Yaskawa INFORM job: apremTRJ0.JBI

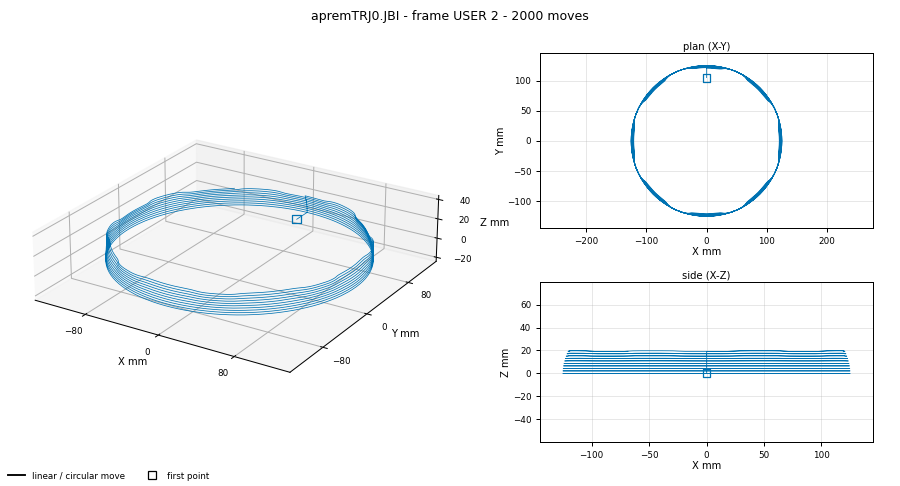
[picture p0: tool path of apremTRJ0.JBI in frame USER 2, 2000 of 2000 moves have a stored position in this frame; points joined in program order, loops and branches not executed]
/JOB
//NAME apremTRJ0
//POS
///NPOS 2000,0,0,0,0,0
///USER 2
///TOOL 1
///POSTYPE USER
///RECTAN
///RCONF 1,0,0,0,0,0,0,0,0,0,0,0,0,0,0,0,0,0,0,0,0,0,0,0
C00000=0.000,105.000,0.000,-180.0000,0.0000,0.0000
C00001=0.000,125.000,0.000,-180.0000,0.0000,0.0000
C00002=7.240,124.790,0.000,-180.0000,-0.0000,0.0000
C00003=13.736,124.243,0.000,-180.0000,-0.0000,0.0000
C00004=19.454,123.477,0.000,-180.0000,-0.0000,0.0000
C00005=23.373,122.796,0.000,-180.0000,-0.0000,0.0000
C00006=26.068,122.252,0.000,-180.0000,-0.0000,0.0000
C00007=28.242,121.768,0.000,-180.0000,-0.0000,0.0000
C00008=30.439,121.237,0.000,-180.0000,-0.0000,0.0000
C00009=33.187,120.514,0.000,-180.0000,-0.0000,0.0000
C00010=36.560,119.534,0.000,-180.0000,-0.0000,0.0000
C00011=40.117,118.388,0.000,-180.0000,-0.0000,0.0000
C00012=43.423,117.215,0.000,-180.0000,-0.0000,0.0000
C00013=46.401,116.069,0.000,-180.0000,-0.0000,0.0000
C00014=49.262,114.884,0.000,-180.0000,-0.0000,0.0000
C00015=52.179,113.589,0.000,-180.0000,-0.0000,0.0000
C00016=55.346,112.080,0.000,180.0000,0.0000,0.0000
C00017=58.672,110.375,0.000,180.0000,0.0000,0.0000
C00018=61.749,108.683,0.000,-180.0000,-0.0000,0.0000
C00019=64.204,107.252,0.000,-180.0000,-0.0000,0.0000
C00020=66.133,106.073,0.000,-180.0000,-0.0000,0.0000
C00021=68.012,104.878,0.000,-180.0000,-0.0000,0.0000
C00022=70.303,103.357,0.000,-180.0000,-0.0000,0.0000
C00023=73.555,101.068,0.000,-180.0000,-0.0000,0.0000
C00024=78.141,97.566,0.000,-180.0000,-0.0000,0.0000
C00025=83.120,93.359,0.000,-180.0000,-0.0000,0.0000
C00026=88.388,88.388,0.000,-180.0000,-0.0000,0.0000
C00027=93.359,83.120,0.000,-180.0000,-0.0000,0.0000
C00028=97.566,78.141,0.000,-180.0000,-0.0000,0.0000
C00029=101.068,73.555,0.000,180.0000,0.0000,0.0000
C00030=103.357,70.303,0.000,-180.0000,-0.0000,0.0000
C00031=104.878,68.012,0.000,-180.0000,-0.0000,0.0000
C00032=106.073,66.133,0.000,-180.0000,-0.0000,0.0000
C00033=107.252,64.204,0.000,-180.0000,-0.0000,0.0000
C00034=108.683,61.749,0.000,-180.0000,-0.0000,0.0000
C00035=110.375,58.672,0.000,-180.0000,-0.0000,0.0000
C00036=112.080,55.346,0.000,-180.0000,-0.0000,0.0000
C00037=113.589,52.179,0.000,-180.0000,-0.0000,0.0000
C00038=114.884,49.262,0.000,-180.0000,-0.0000,0.0000
C00039=116.069,46.401,0.000,-180.0000,-0.0000,0.0000
C00040=117.215,43.423,0.000,-180.0000,-0.0000,0.0000
C00041=118.388,40.117,0.000,-180.0000,-0.0000,0.0000
C00042=119.534,36.560,0.000,-180.0000,-0.0000,0.0000
C00043=120.514,33.187,0.000,-180.0000,-0.0000,0.0000
C00044=121.237,30.439,0.000,-180.0000,-0.0000,0.0000
C00045=121.768,28.242,0.000,-180.0000,-0.0000,0.0000
C00046=122.252,26.068,0.000,-180.0000,-0.0000,0.0000
C00047=122.796,23.373,0.000,-180.0000,-0.0000,0.0000
C00048=123.477,19.454,0.000,-180.0000,-0.0000,0.0000
C00049=124.243,13.736,0.000,-180.0000,-0.0000,0.0000
C00050=124.790,7.240,0.000,-180.0000,-0.0000,0.0000
C00051=125.000,0.000,0.000,-180.0000,-0.0000,0.0000
C00052=124.790,-7.240,0.000,180.0000,-0.0000,0.0000
C00053=124.243,-13.736,0.000,180.0000,-0.0000,0.0000
C00054=123.477,-19.454,0.000,180.0000,-0.0000,0.0000
C00055=122.796,-23.373,0.000,180.0000,-0.0000,0.0000
C00056=122.252,-26.068,0.000,180.0000,-0.0000,0.0000
C00057=121.768,-28.242,0.000,180.0000,-0.0000,0.0000
C00058=121.237,-30.439,0.000,180.0000,-0.0000,0.0000
C00059=120.514,-33.187,0.000,180.0000,-0.0000,0.0000
C00060=119.534,-36.560,0.000,180.0000,-0.0000,0.0000
C00061=118.388,-40.117,0.000,180.0000,-0.0000,0.0000
C00062=117.215,-43.423,0.000,180.0000,-0.0000,0.0000
C00063=116.069,-46.401,0.000,180.0000,-0.0000,0.0000
C00064=114.884,-49.262,0.000,180.0000,-0.0000,0.0000
C00065=113.589,-52.179,0.000,180.0000,-0.0000,0.0000
C00066=112.080,-55.346,0.000,180.0000,-0.0000,0.0000
C00067=110.375,-58.672,0.000,180.0000,-0.0000,0.0000
C00068=108.683,-61.749,0.000,180.0000,-0.0000,0.0000
C00069=107.252,-64.204,0.000,180.0000,-0.0000,0.0000
C00070=106.073,-66.133,0.000,180.0000,-0.0000,0.0000
C00071=104.878,-68.012,0.000,180.0000,-0.0000,0.0000
C00072=103.357,-70.303,0.000,180.0000,-0.0000,0.0000
C00073=101.068,-73.555,0.000,180.0000,-0.0000,0.0000
C00074=97.566,-78.141,0.000,180.0000,-0.0000,0.0000
C00075=93.359,-83.120,0.000,180.0000,-0.0000,0.0000
C00076=88.388,-88.388,0.000,180.0000,-0.0000,0.0000
C00077=83.120,-93.359,0.000,180.0000,-0.0000,0.0000
C00078=78.141,-97.566,0.000,180.0000,-0.0000,0.0000
C00079=73.555,-101.068,0.000,180.0000,-0.0000,0.0000
C00080=70.303,-103.357,0.000,180.0000,-0.0000,0.0000
C00081=68.012,-104.878,0.000,180.0000,-0.0000,0.0000
C00082=66.133,-106.073,0.000,180.0000,-0.0000,0.0000
C00083=64.204,-107.252,0.000,180.0000,-0.0000,0.0000
C00084=61.749,-108.683,0.000,-180.0000,0.0000,0.0000
C00085=58.672,-110.375,0.000,180.0000,-0.0000,0.0000
C00086=55.346,-112.080,0.000,180.0000,-0.0000,0.0000
C00087=52.179,-113.589,0.000,180.0000,-0.0000,0.0000
C00088=49.262,-114.884,0.000,180.0000,-0.0000,0.0000
C00089=46.401,-116.069,0.000,180.0000,-0.0000,0.0000
C00090=43.423,-117.215,0.000,180.0000,-0.0000,0.0000
C00091=40.117,-118.388,0.000,180.0000,-0.0000,0.0000
C00092=36.560,-119.534,0.000,180.0000,-0.0000,0.0000
C00093=33.187,-120.514,0.000,180.0000,-0.0000,0.0000
C00094=30.439,-121.237,0.000,180.0000,-0.0000,0.0000
C00095=28.242,-121.768,0.000,180.0000,-0.0000,0.0000
C00096=26.068,-122.252,0.000,180.0000,-0.0000,0.0000
C00097=23.373,-122.796,0.000,180.0000,-0.0000,0.0000
C00098=19.454,-123.477,0.000,180.0000,-0.0000,0.0000
C00099=13.736,-124.243,0.000,180.0000,-0.0000,0.0000
C00100=7.240,-124.790,0.000,180.0000,-0.0000,0.0000
C00101=0.000,-125.000,0.000,-180.0000,-0.0000,0.0000
C00102=0.000,-125.000,0.000,-180.0000,-0.0000,0.0000
C00103=-7.240,-124.790,0.000,-180.0000,-0.0000,0.0000
C00104=-13.736,-124.243,0.000,-180.0000,-0.0000,0.0000
C00105=-19.454,-123.477,0.000,-180.0000,-0.0000,0.0000
C00106=-23.373,-122.796,0.000,-180.0000,-0.0000,0.0000
C00107=-26.068,-122.252,0.000,-180.0000,-0.0000,0.0000
C00108=-28.242,-121.768,0.000,-180.0000,-0.0000,0.0000
C00109=-30.439,-121.237,0.000,-180.0000,-0.0000,0.0000
C00110=-33.187,-120.514,0.000,-180.0000,-0.0000,0.0000
C00111=-36.560,-119.534,0.000,-180.0000,-0.0000,0.0000
C00112=-40.117,-118.388,0.000,-180.0000,-0.0000,0.0000
C00113=-43.423,-117.215,0.000,-180.0000,-0.0000,0.0000
C00114=-46.401,-116.069,0.000,-180.0000,-0.0000,0.0000
C00115=-49.262,-114.884,0.000,-180.0000,-0.0000,0.0000
C00116=-52.179,-113.589,0.000,-180.0000,-0.0000,0.0000
C00117=-55.346,-112.080,0.000,-180.0000,-0.0000,0.0000
C00118=-58.672,-110.375,0.000,-180.0000,-0.0000,0.0000
C00119=-61.749,-108.683,0.000,-180.0000,-0.0000,0.0000
C00120=-64.204,-107.252,0.000,-180.0000,-0.0000,0.0000
C00121=-66.133,-106.073,0.000,-180.0000,-0.0000,0.0000
C00122=-68.012,-104.878,0.000,-180.0000,-0.0000,0.0000
C00123=-70.303,-103.357,0.000,-180.0000,-0.0000,0.0000
C00124=-73.555,-101.068,0.000,-180.0000,-0.0000,0.0000
C00125=-78.141,-97.566,0.000,-180.0000,-0.0000,0.0000
C00126=-83.120,-93.359,0.000,-180.0000,-0.0000,0.0000
C00127=-88.388,-88.388,0.000,-180.0000,-0.0000,0.0000
C00128=-93.359,-83.120,0.000,-180.0000,-0.0000,0.0000
C00129=-97.566,-78.141,0.000,-180.0000,-0.0000,0.0000
C00130=-101.068,-73.555,0.000,-180.0000,-0.0000,0.0000
C00131=-103.357,-70.303,0.000,-180.0000,-0.0000,0.0000
C00132=-104.878,-68.012,0.000,-180.0000,-0.0000,0.0000
C00133=-106.073,-66.133,0.000,-180.0000,-0.0000,0.0000
C00134=-107.252,-64.204,0.000,-180.0000,-0.0000,0.0000
C00135=-108.683,-61.749,0.000,-180.0000,-0.0000,0.0000
C00136=-110.375,-58.672,0.000,-180.0000,-0.0000,0.0000
C00137=-112.080,-55.346,0.000,-180.0000,-0.0000,0.0000
C00138=-113.589,-52.179,0.000,180.0000,0.0000,0.0000
C00139=-114.884,-49.262,0.000,180.0000,0.0000,0.0000
C00140=-116.069,-46.401,0.000,-180.0000,-0.0000,0.0000
C00141=-117.215,-43.423,0.000,-180.0000,-0.0000,0.0000
C00142=-118.388,-40.117,0.000,180.0000,0.0000,0.0000
C00143=-119.534,-36.560,0.000,180.0000,0.0000,0.0000
C00144=-120.514,-33.187,0.000,-180.0000,-0.0000,0.0000
C00145=-121.237,-30.439,0.000,-180.0000,-0.0000,0.0000
C00146=-121.768,-28.242,0.000,-180.0000,-0.0000,0.0000
C00147=-122.252,-26.068,0.000,-180.0000,-0.0000,0.0000
C00148=-122.796,-23.373,0.000,-180.0000,-0.0000,0.0000
C00149=-123.477,-19.454,0.000,-180.0000,-0.0000,0.0000
C00150=-124.243,-13.736,0.000,-180.0000,-0.0000,0.0000
C00151=-124.790,-7.240,0.000,-180.0000,-0.0000,0.0000
C00152=-125.000,0.000,0.000,180.0000,0.0000,0.0000
C00153=-124.790,7.240,0.000,-180.0000,0.0000,0.0000
C00154=-124.243,13.736,0.000,-180.0000,0.0000,0.0000
C00155=-123.477,19.454,0.000,-180.0000,0.0000,0.0000
C00156=-122.796,23.373,0.000,-180.0000,0.0000,0.0000
C00157=-122.252,26.068,0.000,-180.0000,0.0000,0.0000
C00158=-121.768,28.242,0.000,-180.0000,0.0000,0.0000
C00159=-121.237,30.439,0.000,-180.0000,0.0000,0.0000
C00160=-120.514,33.187,0.000,-180.0000,0.0000,0.0000
C00161=-119.534,36.560,0.000,-180.0000,0.0000,0.0000
C00162=-118.388,40.117,0.000,-180.0000,0.0000,0.0000
C00163=-117.215,43.423,0.000,-180.0000,0.0000,0.0000
C00164=-116.069,46.401,0.000,-180.0000,0.0000,0.0000
C00165=-114.884,49.262,0.000,-180.0000,0.0000,0.0000
C00166=-113.589,52.179,0.000,-180.0000,0.0000,0.0000
C00167=-112.080,55.346,0.000,-180.0000,0.0000,0.0000
C00168=-110.375,58.672,0.000,-180.0000,0.0000,0.0000
C00169=-108.683,61.749,0.000,-180.0000,0.0000,0.0000
C00170=-107.252,64.204,0.000,-180.0000,0.0000,0.0000
C00171=-106.073,66.133,0.000,-180.0000,0.0000,0.0000
C00172=-104.878,68.012,0.000,-180.0000,0.0000,0.0000
C00173=-103.357,70.303,0.000,-180.0000,0.0000,0.0000
C00174=-101.068,73.555,0.000,-180.0000,0.0000,0.0000
C00175=-97.566,78.141,0.000,-180.0000,0.0000,0.0000
C00176=-93.359,83.120,0.000,-180.0000,0.0000,0.0000
C00177=-88.388,88.388,0.000,-180.0000,0.0000,0.0000
C00178=-83.120,93.359,0.000,-180.0000,0.0000,0.0000
C00179=-78.141,97.566,0.000,-180.0000,0.0000,0.0000
C00180=-73.555,101.068,0.000,-180.0000,0.0000,0.0000
C00181=-70.303,103.357,0.000,-180.0000,0.0000,0.0000
C00182=-68.012,104.878,0.000,-180.0000,0.0000,0.0000
C00183=-66.133,106.073,0.000,-180.0000,0.0000,0.0000
C00184=-64.204,107.252,0.000,-180.0000,0.0000,0.0000
C00185=-61.749,108.683,0.000,-180.0000,0.0000,0.0000
C00186=-58.672,110.375,0.000,-180.0000,0.0000,0.0000
C00187=-55.346,112.080,0.000,-180.0000,0.0000,0.0000
C00188=-52.179,113.589,0.000,-180.0000,0.0000,0.0000
C00189=-49.262,114.884,0.000,-180.0000,0.0000,0.0000
C00190=-46.401,116.069,0.000,-180.0000,0.0000,0.0000
C00191=-43.423,117.215,0.000,-180.0000,0.0000,0.0000
C00192=-40.117,118.388,0.000,-180.0000,0.0000,0.0000
C00193=-36.560,119.534,0.000,-180.0000,0.0000,0.0000
C00194=-33.187,120.514,0.000,-180.0000,0.0000,0.0000
C00195=-30.439,121.237,0.000,-180.0000,0.0000,0.0000
C00196=-28.242,121.768,0.000,-180.0000,0.0000,0.0000
C00197=-26.068,122.252,0.000,-180.0000,0.0000,0.0000
C00198=-23.373,122.796,0.000,-180.0000,0.0000,0.0000
C00199=-19.454,123.477,0.000,-180.0000,0.0000,0.0000
C00200=-13.736,124.243,0.000,-180.0000,0.0000,0.0000
C00201=-7.240,124.790,0.000,-180.0000,0.0000,0.0000
C00202=0.000,125.000,0.000,-180.0000,0.0000,0.0000
C00203=0.000,124.937,2.199,-176.7359,0.0000,0.0000
C00204=7.234,124.727,2.199,-176.7395,-0.1900,0.0000
C00205=13.726,124.181,2.199,-176.7605,-0.3579,0.0000
C00206=19.443,123.417,2.199,-176.9022,-0.4857,0.0000
C00207=23.359,122.743,2.199,-177.2352,-0.5194,0.0000
C00208=26.053,122.209,2.200,-177.7082,-0.4785,0.0000
C00209=28.225,121.736,2.200,-178.2567,-0.3947,0.0000
C00210=30.422,121.217,2.200,-178.8064,-0.2941,0.0000
C00211=33.169,120.504,2.200,-179.2794,-0.1963,0.0000
C00212=36.543,119.532,2.200,-179.6554,-0.1047,0.0000
C00213=40.104,118.390,2.200,-179.9022,-0.0330,0.0000
C00214=43.415,117.218,2.200,-179.9844,-0.0058,0.0000
C00215=46.399,116.070,2.200,-179.9982,-0.0007,0.0000
C00216=49.265,114.882,2.200,-179.9982,-0.0008,0.0000
C00217=52.187,113.585,2.200,-179.9849,-0.0069,0.0000
C00218=55.357,112.072,2.200,-179.9075,-0.0458,0.0000
C00219=58.682,110.361,2.200,-179.6823,-0.1696,0.0000
C00220=61.755,108.663,2.200,-179.3516,-0.3707,0.0000
C00221=64.202,107.225,2.200,-178.9481,-0.6362,0.0000
C00222=66.122,106.039,2.200,-178.4882,-0.9539,0.0000
C00223=67.993,104.837,2.200,-178.0410,-1.2829,0.0000
C00224=70.275,103.309,2.199,-177.6774,-1.5889,0.0000
C00225=73.521,101.017,2.199,-177.4656,-1.8485,0.0000
C00226=78.103,97.515,2.199,-177.4554,-2.0392,0.0000
C00227=83.080,93.311,2.199,-177.5592,-2.1726,0.0000
C00228=88.344,88.344,2.199,-177.6906,-2.3094,0.0000
C00229=93.311,83.080,2.199,-177.8274,-2.4408,0.0000
C00230=97.515,78.103,2.199,-177.9608,-2.5446,0.0000
C00231=101.017,73.521,2.199,-178.1515,-2.5344,0.0000
C00232=103.309,70.275,2.199,-178.4111,-2.3226,0.0000
C00233=104.837,67.993,2.200,-178.7171,-1.9590,0.0000
C00234=106.039,66.122,2.200,-179.0461,-1.5118,0.0000
C00235=107.225,64.202,2.200,-179.3638,-1.0519,0.0000
C00236=108.663,61.755,2.200,-179.6293,-0.6484,0.0000
C00237=110.361,58.682,2.200,-179.8304,-0.3177,0.0000
C00238=112.072,55.357,2.200,-179.9542,-0.0925,0.0000
C00239=113.585,52.187,2.200,-179.9931,-0.0151,0.0000
C00240=114.882,49.265,2.200,-179.9992,-0.0018,0.0000
C00241=116.070,46.399,2.200,-179.9993,-0.0018,0.0000
C00242=117.218,43.415,2.200,-179.9942,-0.0156,0.0000
C00243=118.390,40.104,2.200,-179.9670,-0.0978,0.0000
C00244=119.532,36.543,2.200,-179.8953,-0.3446,0.0000
C00245=120.504,33.169,2.200,-179.8037,-0.7206,0.0000
C00246=121.217,30.422,2.200,-179.7059,-1.1936,0.0000
C00247=121.736,28.225,2.200,-179.6053,-1.7433,0.0000
C00248=122.209,26.053,2.200,-179.5215,-2.2918,0.0000
C00249=122.743,23.359,2.199,-179.4806,-2.7648,0.0000
C00250=123.417,19.443,2.199,-179.5143,-3.0978,0.0000
C00251=124.181,13.726,2.199,-179.6421,-3.2395,0.0000
C00252=124.727,7.234,2.199,-179.8100,-3.2605,0.0000
C00253=124.937,0.000,2.199,180.0000,-3.2641,0.0000
C00254=124.727,-7.234,2.199,179.8100,-3.2604,0.0000
C00255=124.181,-13.726,2.199,179.6421,-3.2395,0.0000
C00256=123.417,-19.443,2.199,179.5143,-3.0978,0.0000
C00257=122.743,-23.359,2.199,179.4806,-2.7648,0.0000
C00258=122.209,-26.053,2.200,179.5215,-2.2918,0.0000
C00259=121.736,-28.225,2.200,179.6053,-1.7433,0.0000
C00260=121.217,-30.422,2.200,179.7059,-1.1936,0.0000
C00261=120.504,-33.169,2.200,179.8037,-0.7206,0.0000
C00262=119.532,-36.543,2.200,179.8953,-0.3446,0.0000
C00263=118.390,-40.104,2.200,179.9670,-0.0978,0.0000
C00264=117.218,-43.415,2.200,179.9942,-0.0156,0.0000
C00265=116.070,-46.399,2.200,179.9993,-0.0018,0.0000
C00266=114.882,-49.265,2.200,179.9992,-0.0018,0.0000
C00267=113.585,-52.187,2.200,179.9931,-0.0151,0.0000
C00268=112.072,-55.357,2.200,179.9542,-0.0925,0.0000
C00269=110.361,-58.682,2.200,179.8304,-0.3177,0.0000
C00270=108.663,-61.755,2.200,179.6293,-0.6484,0.0000
C00271=107.225,-64.202,2.200,179.3638,-1.0519,0.0000
C00272=106.039,-66.122,2.200,179.0461,-1.5118,0.0000
C00273=104.837,-67.993,2.200,178.7171,-1.9590,0.0000
C00274=103.309,-70.275,2.199,178.4111,-2.3226,0.0000
C00275=101.017,-73.521,2.199,178.1515,-2.5344,0.0000
C00276=97.515,-78.103,2.199,177.9608,-2.5446,0.0000
C00277=93.311,-83.080,2.199,177.8274,-2.4408,0.0000
C00278=88.344,-88.344,2.199,177.6906,-2.3094,0.0000
C00279=83.080,-93.311,2.199,177.5592,-2.1726,0.0000
C00280=78.103,-97.515,2.199,177.4554,-2.0392,0.0000
C00281=73.521,-101.017,2.199,177.4656,-1.8485,0.0000
C00282=70.275,-103.309,2.199,177.6774,-1.5889,0.0000
C00283=67.993,-104.837,2.200,178.0410,-1.2829,0.0000
C00284=66.122,-106.039,2.200,178.4882,-0.9539,0.0000
C00285=64.202,-107.225,2.200,178.9481,-0.6362,0.0000
C00286=61.755,-108.663,2.200,179.3516,-0.3707,0.0000
C00287=58.682,-110.361,2.200,179.6823,-0.1696,0.0000
C00288=55.357,-112.072,2.200,179.9075,-0.0458,0.0000
C00289=52.187,-113.585,2.200,179.9849,-0.0069,0.0000
C00290=49.265,-114.882,2.200,179.9982,-0.0008,0.0000
C00291=46.399,-116.070,2.200,179.9982,-0.0007,0.0000
C00292=43.415,-117.218,2.200,179.9844,-0.0058,0.0000
C00293=40.104,-118.390,2.200,179.9022,-0.0330,0.0000
C00294=36.543,-119.532,2.200,179.6554,-0.1047,0.0000
C00295=33.169,-120.504,2.200,179.2794,-0.1963,0.0000
C00296=30.422,-121.217,2.200,178.8064,-0.2941,0.0000
C00297=28.225,-121.736,2.200,178.2567,-0.3947,0.0000
C00298=26.053,-122.209,2.200,177.7082,-0.4785,0.0000
C00299=23.359,-122.743,2.199,177.2352,-0.5194,0.0000
C00300=19.443,-123.417,2.199,176.9022,-0.4857,0.0000
C00301=13.726,-124.181,2.199,176.7605,-0.3579,0.0000
C00302=7.234,-124.727,2.199,176.7395,-0.1900,0.0000
C00303=0.000,-124.937,2.199,176.7359,0.0000,0.0000
C00304=0.000,-124.937,2.199,176.7359,0.0000,0.0000
C00305=-7.234,-124.727,2.199,176.7396,0.1900,0.0000
C00306=-13.726,-124.181,2.199,176.7605,0.3579,0.0000
C00307=-19.443,-123.417,2.199,176.9022,0.4857,0.0000
C00308=-23.359,-122.743,2.199,177.2352,0.5194,0.0000
C00309=-26.053,-122.209,2.200,177.7082,0.4785,0.0000
C00310=-28.225,-121.736,2.200,178.2567,0.3947,0.0000
C00311=-30.422,-121.217,2.200,178.8064,0.2941,0.0000
C00312=-33.169,-120.504,2.200,179.2794,0.1963,0.0000
C00313=-36.543,-119.532,2.200,179.6554,0.1047,0.0000
C00314=-40.104,-118.390,2.200,179.9022,0.0330,0.0000
C00315=-43.415,-117.218,2.200,179.9844,0.0058,0.0000
C00316=-46.399,-116.070,2.200,179.9982,0.0007,0.0000
C00317=-49.265,-114.882,2.200,179.9982,0.0008,0.0000
C00318=-52.187,-113.585,2.200,179.9849,0.0069,0.0000
C00319=-55.357,-112.072,2.200,179.9075,0.0458,0.0000
C00320=-58.682,-110.361,2.200,179.6823,0.1696,0.0000
C00321=-61.755,-108.663,2.200,179.3516,0.3707,0.0000
C00322=-64.202,-107.225,2.200,178.9481,0.6362,0.0000
C00323=-66.122,-106.039,2.200,178.4882,0.9539,0.0000
C00324=-67.993,-104.837,2.200,178.0410,1.2829,0.0000
C00325=-70.275,-103.309,2.199,177.6774,1.5889,0.0000
C00326=-73.521,-101.017,2.199,177.4656,1.8485,0.0000
C00327=-78.103,-97.515,2.199,177.4554,2.0392,0.0000
C00328=-83.080,-93.311,2.199,177.5592,2.1726,0.0000
C00329=-88.344,-88.344,2.199,177.6906,2.3094,0.0000
C00330=-93.311,-83.080,2.199,177.8274,2.4408,0.0000
C00331=-97.515,-78.103,2.199,177.9608,2.5446,0.0000
C00332=-101.017,-73.521,2.199,178.1515,2.5344,0.0000
C00333=-103.309,-70.275,2.199,178.4111,2.3226,0.0000
C00334=-104.837,-67.993,2.200,178.7171,1.9590,0.0000
C00335=-106.039,-66.122,2.200,179.0461,1.5118,0.0000
C00336=-107.225,-64.202,2.200,179.3638,1.0519,0.0000
C00337=-108.663,-61.755,2.200,179.6293,0.6484,0.0000
C00338=-110.361,-58.682,2.200,179.8304,0.3177,0.0000
C00339=-112.072,-55.357,2.200,179.9542,0.0925,0.0000
C00340=-113.585,-52.187,2.200,179.9931,0.0151,0.0000
C00341=-114.882,-49.265,2.200,179.9992,0.0018,0.0000
C00342=-116.070,-46.399,2.200,179.9993,0.0018,0.0000
C00343=-117.218,-43.415,2.200,179.9942,0.0156,0.0000
C00344=-118.390,-40.104,2.200,179.9670,0.0978,0.0000
C00345=-119.532,-36.543,2.200,179.8953,0.3446,0.0000
C00346=-120.504,-33.169,2.200,179.8037,0.7206,0.0000
C00347=-121.217,-30.422,2.200,179.7059,1.1936,0.0000
C00348=-121.736,-28.225,2.200,179.6053,1.7433,0.0000
C00349=-122.209,-26.053,2.200,179.5215,2.2918,0.0000
C00350=-122.743,-23.359,2.199,179.4806,2.7648,0.0000
C00351=-123.417,-19.443,2.199,179.5143,3.0978,0.0000
C00352=-124.181,-13.726,2.199,179.6421,3.2395,0.0000
C00353=-124.727,-7.234,2.199,179.8100,3.2605,0.0000
C00354=-124.937,0.000,2.199,-180.0000,3.2641,0.0000
C00355=-124.727,7.234,2.199,-179.8100,3.2604,0.0000
C00356=-124.181,13.726,2.199,-179.6421,3.2395,0.0000
C00357=-123.417,19.443,2.199,-179.5143,3.0978,0.0000
C00358=-122.743,23.359,2.199,-179.4806,2.7648,0.0000
C00359=-122.209,26.053,2.200,-179.5215,2.2918,0.0000
C00360=-121.736,28.225,2.200,-179.6053,1.7433,0.0000
C00361=-121.217,30.422,2.200,-179.7059,1.1936,0.0000
C00362=-120.504,33.169,2.200,-179.8037,0.7206,0.0000
C00363=-119.532,36.543,2.200,-179.8953,0.3446,0.0000
C00364=-118.390,40.104,2.200,-179.9670,0.0978,0.0000
C00365=-117.218,43.415,2.200,-179.9942,0.0156,0.0000
C00366=-116.070,46.399,2.200,-179.9993,0.0018,0.0000
C00367=-114.882,49.265,2.200,-179.9992,0.0018,0.0000
C00368=-113.585,52.187,2.200,-179.9931,0.0151,0.0000
C00369=-112.072,55.357,2.200,-179.9542,0.0925,0.0000
C00370=-110.361,58.682,2.200,-179.8304,0.3177,0.0000
C00371=-108.663,61.755,2.200,-179.6293,0.6484,0.0000
C00372=-107.225,64.202,2.200,-179.3638,1.0519,0.0000
C00373=-106.039,66.122,2.200,-179.0461,1.5118,0.0000
C00374=-104.837,67.993,2.200,-178.7171,1.9590,0.0000
C00375=-103.309,70.275,2.199,-178.4111,2.3226,0.0000
C00376=-101.017,73.521,2.199,-178.1515,2.5344,0.0000
C00377=-97.515,78.103,2.199,-177.9608,2.5446,0.0000
C00378=-93.311,83.080,2.199,-177.8274,2.4408,0.0000
C00379=-88.344,88.344,2.199,-177.6906,2.3094,0.0000
C00380=-83.080,93.311,2.199,-177.5592,2.1726,0.0000
C00381=-78.103,97.515,2.199,-177.4554,2.0392,0.0000
C00382=-73.521,101.017,2.199,-177.4656,1.8485,0.0000
C00383=-70.275,103.309,2.199,-177.6774,1.5889,0.0000
C00384=-67.993,104.837,2.200,-178.0410,1.2829,0.0000
C00385=-66.122,106.039,2.200,-178.4882,0.9539,0.0000
C00386=-64.202,107.225,2.200,-178.9481,0.6362,0.0000
C00387=-61.755,108.663,2.200,-179.3516,0.3707,0.0000
C00388=-58.682,110.361,2.200,-179.6823,0.1696,0.0000
C00389=-55.357,112.072,2.200,-179.9075,0.0458,0.0000
C00390=-52.187,113.585,2.200,-179.9849,0.0069,0.0000
C00391=-49.265,114.882,2.200,-179.9982,0.0008,0.0000
C00392=-46.399,116.070,2.200,-179.9982,0.0007,0.0000
C00393=-43.415,117.218,2.200,-179.9844,0.0058,0.0000
C00394=-40.104,118.390,2.200,-179.9022,0.0330,0.0000
C00395=-36.543,119.532,2.200,-179.6554,0.1047,0.0000
C00396=-33.169,120.504,2.200,-179.2794,0.1963,0.0000
C00397=-30.422,121.217,2.200,-178.8064,0.2941,0.0000
C00398=-28.225,121.736,2.200,-178.2567,0.3947,0.0000
C00399=-26.053,122.209,2.200,-177.7082,0.4785,0.0000
C00400=-23.359,122.743,2.199,-177.2352,0.5194,0.0000
C00401=-19.443,123.417,2.199,-176.9022,0.4857,0.0000
C00402=-13.726,124.181,2.199,-176.7605,0.3579,0.0000
C00403=-7.234,124.727,2.199,-176.7396,0.1900,0.0000
C00404=0.000,124.937,2.199,-176.7359,0.0000,0.0000
C00405=0.000,124.751,4.391,-173.6081,0.0000,0.0000
C00406=7.217,124.542,4.391,-173.6153,-0.3730,0.0000
C00407=13.697,123.997,4.391,-173.6559,-0.7003,0.0000
C00408=19.408,123.242,4.392,-173.9305,-0.9378,0.0000
C00409=23.317,122.588,4.393,-174.5780,-0.9792,0.0000
C00410=26.007,122.082,4.395,-175.5036,-0.8805,0.0000
C00411=28.178,121.643,4.397,-176.5830,-0.7191,0.0000
C00412=30.372,121.157,4.398,-177.6658,-0.5439,0.0000
C00413=33.115,120.475,4.399,-178.5947,-0.3708,0.0000
C00414=36.492,119.526,4.399,-179.3309,-0.1993,0.0000
C00415=40.064,118.397,4.400,-179.8118,-0.0629,0.0000
C00416=43.390,117.226,4.400,-179.9699,-0.0111,0.0000
C00417=46.390,116.073,4.400,-179.9965,-0.0014,0.0000
C00418=49.273,114.879,4.400,-179.9965,-0.0015,0.0000
C00419=52.210,113.573,4.400,-179.9709,-0.0134,0.0000
C00420=55.390,112.049,4.400,-179.8224,-0.0886,0.0000
C00421=58.714,110.321,4.399,-179.3860,-0.3322,0.0000
C00422=61.773,108.604,4.399,-178.7441,-0.7317,0.0000
C00423=64.195,107.147,4.398,-177.9648,-1.2666,0.0000
C00424=66.090,105.939,4.397,-177.0750,-1.9098,0.0000
C00425=67.935,104.715,4.395,-176.1970,-2.5616,0.0000
C00426=70.195,103.171,4.393,-175.4716,-3.1498,0.0000
C00427=73.422,100.869,4.392,-175.0413,-3.6398,0.0000
C00428=77.994,97.365,4.391,-175.0131,-4.0027,0.0000
C00429=82.961,93.168,4.391,-175.2140,-4.2618,0.0000
C00430=88.212,88.212,4.391,-175.4709,-4.5291,0.0000
C00431=93.168,82.961,4.391,-175.7382,-4.7860,0.0000
C00432=97.365,77.994,4.391,-175.9973,-4.9870,0.0000
C00433=100.869,73.422,4.392,-176.3602,-4.9586,0.0000
C00434=103.171,70.195,4.393,-176.8502,-4.5284,0.0000
C00435=104.715,67.935,4.395,-177.4384,-3.8030,0.0000
C00436=105.939,66.090,4.397,-178.0902,-2.9250,0.0000
C00437=107.147,64.195,4.398,-178.7334,-2.0352,0.0000
C00438=108.604,61.773,4.399,-179.2683,-1.2559,0.0000
C00439=110.321,58.714,4.399,-179.6678,-0.6140,0.0000
C00440=112.049,55.390,4.400,-179.9114,-0.1776,0.0000
C00441=113.573,52.210,4.400,-179.9866,-0.0291,0.0000
C00442=114.879,49.273,4.400,-179.9985,-0.0035,0.0000
C00443=116.073,46.390,4.400,-179.9986,-0.0035,0.0000
C00444=117.226,43.390,4.400,-179.9889,-0.0301,0.0000
C00445=118.397,40.064,4.400,-179.9371,-0.1882,0.0000
C00446=119.526,36.492,4.399,-179.8007,-0.6691,0.0000
C00447=120.475,33.115,4.399,-179.6292,-1.4053,0.0000
C00448=121.157,30.372,4.398,-179.4561,-2.3342,0.0000
C00449=121.643,28.178,4.397,-179.2809,-3.4170,0.0000
C00450=122.082,26.007,4.395,-179.1195,-4.4964,0.0000
C00451=122.588,23.317,4.393,-179.0208,-5.4220,0.0000
C00452=123.242,19.408,4.392,-179.0622,-6.0695,0.0000
C00453=123.997,13.697,4.391,-179.2997,-6.3441,0.0000
C00454=124.542,7.217,4.391,-179.6270,-6.3847,0.0000
C00455=124.751,0.000,4.391,180.0000,-6.3919,0.0000
C00456=124.542,-7.217,4.391,179.6271,-6.3846,0.0000
C00457=123.997,-13.697,4.391,179.2997,-6.3441,0.0000
C00458=123.242,-19.408,4.392,179.0622,-6.0694,0.0000
C00459=122.588,-23.317,4.393,179.0208,-5.4220,0.0000
C00460=122.082,-26.007,4.395,179.1195,-4.4964,0.0000
C00461=121.643,-28.178,4.397,179.2809,-3.4170,0.0000
C00462=121.157,-30.372,4.398,179.4561,-2.3342,0.0000
C00463=120.475,-33.115,4.399,179.6292,-1.4053,0.0000
C00464=119.526,-36.492,4.399,179.8007,-0.6691,0.0000
C00465=118.397,-40.064,4.400,179.9371,-0.1882,0.0000
C00466=117.226,-43.390,4.400,179.9889,-0.0301,0.0000
C00467=116.073,-46.390,4.400,179.9986,-0.0035,0.0000
C00468=114.879,-49.273,4.400,179.9985,-0.0035,0.0000
C00469=113.573,-52.210,4.400,179.9866,-0.0291,0.0000
C00470=112.049,-55.390,4.400,179.9114,-0.1776,0.0000
C00471=110.321,-58.714,4.399,179.6678,-0.6140,0.0000
C00472=108.604,-61.773,4.399,179.2683,-1.2559,0.0000
C00473=107.147,-64.195,4.398,178.7334,-2.0352,0.0000
C00474=105.939,-66.090,4.397,178.0902,-2.9250,0.0000
C00475=104.715,-67.935,4.395,177.4384,-3.8030,0.0000
C00476=103.171,-70.195,4.393,176.8502,-4.5284,0.0000
C00477=100.869,-73.422,4.392,176.3602,-4.9587,0.0000
C00478=97.365,-77.994,4.391,175.9973,-4.9869,0.0000
C00479=93.168,-82.961,4.391,175.7382,-4.7860,0.0000
C00480=88.212,-88.212,4.391,175.4709,-4.5291,0.0000
C00481=82.961,-93.168,4.391,175.2140,-4.2618,0.0000
C00482=77.994,-97.365,4.391,175.0130,-4.0027,0.0000
C00483=73.422,-100.869,4.392,175.0414,-3.6398,0.0000
C00484=70.195,-103.171,4.393,175.4716,-3.1498,0.0000
C00485=67.935,-104.715,4.395,176.1970,-2.5616,0.0000
C00486=66.090,-105.939,4.397,177.0750,-1.9098,0.0000
C00487=64.195,-107.147,4.398,177.9648,-1.2666,0.0000
C00488=61.773,-108.604,4.399,178.7441,-0.7317,0.0000
C00489=58.714,-110.321,4.399,179.3860,-0.3322,0.0000
C00490=55.390,-112.049,4.400,179.8224,-0.0886,0.0000
C00491=52.210,-113.573,4.400,179.9709,-0.0134,0.0000
C00492=49.273,-114.879,4.400,179.9965,-0.0015,0.0000
C00493=46.390,-116.073,4.400,179.9965,-0.0014,0.0000
C00494=43.390,-117.226,4.400,179.9699,-0.0111,0.0000
C00495=40.064,-118.397,4.400,179.8118,-0.0629,0.0000
C00496=36.492,-119.526,4.399,179.3309,-0.1993,0.0000
C00497=33.115,-120.475,4.399,178.5947,-0.3708,0.0000
C00498=30.372,-121.157,4.398,177.6658,-0.5439,0.0000
C00499=28.178,-121.643,4.397,176.5830,-0.7191,0.0000
C00500=26.007,-122.082,4.395,175.5036,-0.8805,0.0000
C00501=23.317,-122.588,4.393,174.5780,-0.9792,0.0000
C00502=19.408,-123.242,4.392,173.9305,-0.9378,0.0000
C00503=13.697,-123.997,4.391,173.6559,-0.7003,0.0000
C00504=7.217,-124.542,4.391,173.6153,-0.3730,0.0000
C00505=0.000,-124.751,4.391,173.6081,0.0000,0.0000
C00506=0.000,-124.751,4.391,173.6081,0.0000,0.0000
C00507=-7.217,-124.542,4.391,173.6154,0.3729,0.0000
C00508=-13.697,-123.997,4.391,173.6559,0.7003,0.0000
C00509=-19.408,-123.242,4.392,173.9306,0.9378,0.0000
C00510=-23.317,-122.588,4.393,174.5780,0.9792,0.0000
C00511=-26.007,-122.082,4.395,175.5036,0.8805,0.0000
C00512=-28.178,-121.643,4.397,176.5830,0.7191,0.0000
C00513=-30.372,-121.157,4.398,177.6658,0.5439,0.0000
C00514=-33.115,-120.475,4.399,178.5947,0.3708,0.0000
C00515=-36.492,-119.526,4.399,179.3309,0.1993,0.0000
C00516=-40.064,-118.397,4.400,179.8118,0.0629,0.0000
C00517=-43.390,-117.226,4.400,179.9699,0.0111,0.0000
C00518=-46.390,-116.073,4.400,179.9965,0.0014,0.0000
C00519=-49.273,-114.879,4.400,179.9965,0.0015,0.0000
C00520=-52.210,-113.573,4.400,179.9709,0.0134,0.0000
C00521=-55.390,-112.049,4.400,179.8224,0.0886,0.0000
C00522=-58.714,-110.321,4.399,179.3860,0.3322,0.0000
C00523=-61.773,-108.604,4.399,178.7441,0.7317,0.0000
C00524=-64.195,-107.147,4.398,177.9648,1.2666,0.0000
C00525=-66.090,-105.939,4.397,177.0750,1.9098,0.0000
C00526=-67.935,-104.715,4.395,176.1970,2.5616,0.0000
C00527=-70.195,-103.171,4.393,175.4716,3.1498,0.0000
C00528=-73.422,-100.869,4.392,175.0413,3.6398,0.0000
C00529=-77.994,-97.365,4.391,175.0131,4.0027,0.0000
C00530=-82.961,-93.168,4.391,175.2140,4.2618,0.0000
C00531=-88.212,-88.212,4.391,175.4709,4.5291,0.0000
C00532=-93.168,-82.961,4.391,175.7382,4.7860,0.0000
C00533=-97.365,-77.994,4.391,175.9973,4.9870,0.0000
C00534=-100.869,-73.422,4.392,176.3602,4.9586,0.0000
C00535=-103.171,-70.195,4.393,176.8502,4.5284,0.0000
C00536=-104.715,-67.935,4.395,177.4384,3.8030,0.0000
C00537=-105.939,-66.090,4.397,178.0902,2.9250,0.0000
C00538=-107.147,-64.195,4.398,178.7334,2.0352,0.0000
C00539=-108.604,-61.773,4.399,179.2683,1.2559,0.0000
C00540=-110.321,-58.714,4.399,179.6678,0.6140,0.0000
C00541=-112.049,-55.390,4.400,179.9114,0.1776,0.0000
C00542=-113.573,-52.210,4.400,179.9866,0.0291,0.0000
C00543=-114.879,-49.273,4.400,179.9985,0.0035,0.0000
C00544=-116.073,-46.390,4.400,179.9986,0.0035,0.0000
C00545=-117.226,-43.390,4.400,179.9889,0.0301,0.0000
C00546=-118.397,-40.064,4.400,179.9371,0.1882,0.0000
C00547=-119.526,-36.492,4.399,179.8007,0.6691,0.0000
C00548=-120.475,-33.115,4.399,179.6292,1.4053,0.0000
C00549=-121.157,-30.372,4.398,179.4561,2.3342,0.0000
C00550=-121.643,-28.178,4.397,179.2809,3.4170,0.0000
C00551=-122.082,-26.007,4.395,179.1195,4.4964,0.0000
C00552=-122.588,-23.317,4.393,179.0208,5.4220,0.0000
C00553=-123.242,-19.408,4.392,179.0622,6.0695,0.0000
C00554=-123.997,-13.697,4.391,179.2997,6.3441,0.0000
C00555=-124.542,-7.217,4.391,179.6270,6.3847,0.0000
C00556=-124.751,0.000,4.391,-180.0000,6.3919,0.0000
C00557=-124.542,7.217,4.391,-179.6271,6.3846,0.0000
C00558=-123.997,13.697,4.391,-179.2997,6.3441,0.0000
C00559=-123.242,19.408,4.392,-179.0622,6.0694,0.0000
C00560=-122.588,23.317,4.393,-179.0208,5.4220,0.0000
C00561=-122.082,26.007,4.395,-179.1195,4.4964,0.0000
C00562=-121.643,28.178,4.397,-179.2809,3.4170,0.0000
C00563=-121.157,30.372,4.398,-179.4561,2.3342,0.0000
C00564=-120.475,33.115,4.399,-179.6292,1.4053,0.0000
C00565=-119.526,36.492,4.399,-179.8007,0.6691,0.0000
C00566=-118.397,40.064,4.400,-179.9371,0.1882,0.0000
C00567=-117.226,43.390,4.400,-179.9889,0.0301,0.0000
C00568=-116.073,46.390,4.400,-179.9986,0.0035,0.0000
C00569=-114.879,49.273,4.400,-179.9985,0.0035,0.0000
C00570=-113.573,52.210,4.400,-179.9866,0.0291,0.0000
C00571=-112.049,55.390,4.400,-179.9114,0.1776,0.0000
C00572=-110.321,58.714,4.399,-179.6678,0.6140,0.0000
C00573=-108.604,61.773,4.399,-179.2683,1.2559,0.0000
C00574=-107.147,64.195,4.398,-178.7334,2.0352,0.0000
C00575=-105.939,66.090,4.397,-178.0902,2.9250,0.0000
C00576=-104.715,67.935,4.395,-177.4384,3.8030,0.0000
C00577=-103.171,70.195,4.393,-176.8502,4.5284,0.0000
C00578=-100.869,73.422,4.392,-176.3602,4.9587,0.0000
C00579=-97.365,77.994,4.391,-175.9973,4.9869,0.0000
C00580=-93.168,82.961,4.391,-175.7382,4.7860,0.0000
C00581=-88.212,88.212,4.391,-175.4709,4.5291,0.0000
C00582=-82.961,93.168,4.391,-175.2140,4.2618,0.0000
C00583=-77.994,97.365,4.391,-175.0130,4.0027,0.0000
C00584=-73.422,100.869,4.392,-175.0414,3.6398,0.0000
C00585=-70.195,103.171,4.393,-175.4716,3.1498,0.0000
C00586=-67.935,104.715,4.395,-176.1970,2.5616,0.0000
C00587=-66.090,105.939,4.397,-177.0750,1.9098,0.0000
C00588=-64.195,107.147,4.398,-177.9648,1.2666,0.0000
C00589=-61.773,108.604,4.399,-178.7441,0.7317,0.0000
C00590=-58.714,110.321,4.399,-179.3860,0.3322,0.0000
C00591=-55.390,112.049,4.400,-179.8224,0.0886,0.0000
C00592=-52.210,113.573,4.400,-179.9709,0.0134,0.0000
C00593=-49.273,114.879,4.400,-179.9965,0.0015,0.0000
C00594=-46.390,116.073,4.400,-179.9965,0.0014,0.0000
C00595=-43.390,117.226,4.400,-179.9699,0.0111,0.0000
C00596=-40.064,118.397,4.400,-179.8118,0.0629,0.0000
C00597=-36.492,119.526,4.399,-179.3309,0.1993,0.0000
C00598=-33.115,120.475,4.399,-178.5947,0.3708,0.0000
C00599=-30.372,121.157,4.398,-177.6658,0.5439,0.0000
C00600=-28.178,121.643,4.397,-176.5830,0.7191,0.0000
C00601=-26.007,122.082,4.395,-175.5036,0.8805,0.0000
C00602=-23.317,122.588,4.393,-174.5780,0.9792,0.0000
C00603=-19.408,123.242,4.392,-173.9306,0.9378,0.0000
C00604=-13.697,123.997,4.391,-173.6559,0.7003,0.0000
C00605=-7.217,124.542,4.391,-173.6154,0.3729,0.0000
C00606=0.000,124.751,4.391,-173.6081,0.0000,0.0000
C00607=0.000,124.449,6.570,-170.6405,0.0000,0.0000
C00608=7.190,124.241,6.570,-170.6509,-0.5483,0.0000
C00609=13.651,123.699,6.570,-170.7093,-1.0235,0.0000
C00610=19.352,122.957,6.573,-171.1043,-1.3408,0.0000
C00611=23.250,122.335,6.578,-172.0415,-1.3416,0.0000
C00612=25.933,121.876,6.584,-173.3969,-1.1521,0.0000
C00613=28.099,121.490,6.590,-174.9904,-0.9229,0.0000
C00614=30.290,121.060,6.595,-176.5889,-0.7201,0.0000
C00615=33.027,120.427,6.597,-177.9550,-0.5107,0.0000
C00616=36.409,119.516,6.598,-179.0332,-0.2787,0.0000
C00617=39.998,118.409,6.599,-179.7323,-0.0880,0.0000
C00618=43.349,117.240,6.599,-179.9569,-0.0159,0.0000
C00619=46.376,116.078,6.600,-179.9949,-0.0020,0.0000
C00620=49.287,114.873,6.600,-179.9950,-0.0021,0.0000
C00621=52.249,113.553,6.599,-179.9583,-0.0192,0.0000
C00622=55.445,112.011,6.599,-179.7485,-0.1271,0.0000
C00623=58.765,110.256,6.598,-179.1193,-0.4866,0.0000
C00624=61.801,108.508,6.597,-178.1928,-1.0854,0.0000
C00625=64.184,107.020,6.595,-177.0785,-1.9049,0.0000
C00626=66.037,105.776,6.590,-175.8035,-2.8963,0.0000
C00627=67.842,104.516,6.584,-174.5122,-3.8692,0.0000
C00628=70.064,102.945,6.578,-173.4163,-4.7046,0.0000
C00629=73.260,100.628,6.573,-172.7494,-5.3772,0.0000
C00630=77.816,97.121,6.570,-172.6884,-5.8831,0.0000
C00631=82.768,92.936,6.570,-172.9775,-6.2574,0.0000
C00632=87.999,87.999,6.570,-173.3523,-6.6477,0.0000
C00633=92.936,82.768,6.570,-173.7426,-7.0224,0.0000
C00634=97.121,77.816,6.570,-174.1168,-7.3116,0.0000
C00635=100.628,73.260,6.573,-174.6229,-7.2506,0.0000
C00636=102.945,70.064,6.578,-175.2954,-6.5837,0.0000
C00637=104.516,67.842,6.584,-176.1308,-5.4878,0.0000
C00638=105.776,66.037,6.590,-177.1037,-4.1965,0.0000
C00639=107.020,64.184,6.595,-178.0951,-2.9215,0.0000
C00640=108.508,61.801,6.597,-178.9146,-1.8072,0.0000
C00641=110.256,58.765,6.598,-179.5134,-0.8807,0.0000
C00642=112.011,55.445,6.599,-179.8729,-0.2515,0.0000
C00643=113.553,52.249,6.599,-179.9808,-0.0417,0.0000
C00644=114.873,49.287,6.600,-179.9979,-0.0050,0.0000
C00645=116.078,46.376,6.600,-179.9980,-0.0051,0.0000
C00646=117.240,43.349,6.599,-179.9841,-0.0431,0.0000
C00647=118.409,39.998,6.599,-179.9120,-0.2677,0.0000
C00648=119.516,36.409,6.598,-179.7213,-0.9668,0.0000
C00649=120.427,33.027,6.597,-179.4893,-2.0450,0.0000
C00650=121.060,30.290,6.595,-179.2799,-3.4111,0.0000
C00651=121.490,28.099,6.590,-179.0771,-5.0096,0.0000
C00652=121.876,25.933,6.584,-178.8479,-6.6031,0.0000
C00653=122.335,23.250,6.578,-178.6584,-7.9585,0.0000
C00654=122.957,19.352,6.573,-178.6592,-8.8957,0.0000
C00655=123.699,13.651,6.570,-178.9765,-9.2907,0.0000
C00656=124.241,7.190,6.570,-179.4517,-9.3491,0.0000
C00657=124.449,0.000,6.570,180.0000,-9.3595,0.0000
C00658=124.241,-7.190,6.570,179.4517,-9.3491,0.0000
C00659=123.699,-13.651,6.570,178.9765,-9.2907,0.0000
C00660=122.957,-19.352,6.573,178.6592,-8.8957,0.0000
C00661=122.335,-23.250,6.578,178.6584,-7.9585,0.0000
C00662=121.876,-25.933,6.584,178.8479,-6.6031,0.0000
C00663=121.490,-28.099,6.590,179.0771,-5.0096,0.0000
C00664=121.060,-30.290,6.595,179.2799,-3.4111,0.0000
C00665=120.427,-33.027,6.597,179.4893,-2.0450,0.0000
C00666=119.516,-36.409,6.598,179.7213,-0.9668,0.0000
C00667=118.409,-39.998,6.599,179.9120,-0.2677,0.0000
C00668=117.240,-43.349,6.599,179.9841,-0.0431,0.0000
C00669=116.078,-46.376,6.600,179.9980,-0.0051,0.0000
C00670=114.873,-49.287,6.600,179.9979,-0.0050,0.0000
C00671=113.553,-52.249,6.599,179.9808,-0.0417,0.0000
C00672=112.011,-55.445,6.599,179.8729,-0.2515,0.0000
C00673=110.256,-58.765,6.598,179.5134,-0.8807,0.0000
C00674=108.508,-61.801,6.597,178.9146,-1.8072,0.0000
C00675=107.020,-64.184,6.595,178.0951,-2.9215,0.0000
C00676=105.776,-66.037,6.590,177.1037,-4.1965,0.0000
C00677=104.516,-67.842,6.584,176.1308,-5.4878,0.0000
C00678=102.945,-70.064,6.578,175.2954,-6.5837,0.0000
C00679=100.628,-73.260,6.573,174.6228,-7.2506,0.0000
C00680=97.121,-77.816,6.570,174.1169,-7.3116,0.0000
C00681=92.936,-82.768,6.570,173.7426,-7.0225,0.0000
C00682=87.999,-87.999,6.570,173.3523,-6.6477,0.0000
C00683=82.768,-92.936,6.570,172.9776,-6.2574,0.0000
C00684=77.816,-97.121,6.570,172.6884,-5.8832,0.0000
C00685=73.260,-100.628,6.573,172.7494,-5.3771,0.0000
C00686=70.064,-102.945,6.578,173.4163,-4.7046,0.0000
C00687=67.842,-104.516,6.584,174.5122,-3.8692,0.0000
C00688=66.037,-105.776,6.590,175.8035,-2.8963,0.0000
C00689=64.184,-107.020,6.595,177.0785,-1.9049,0.0000
C00690=61.801,-108.508,6.597,178.1928,-1.0854,0.0000
C00691=58.765,-110.256,6.598,179.1193,-0.4866,0.0000
C00692=55.445,-112.011,6.599,179.7485,-0.1271,0.0000
C00693=52.249,-113.553,6.599,179.9583,-0.0192,0.0000
C00694=49.287,-114.873,6.600,179.9950,-0.0021,0.0000
C00695=46.376,-116.078,6.600,179.9949,-0.0020,0.0000
C00696=43.349,-117.240,6.599,179.9569,-0.0159,0.0000
C00697=39.998,-118.409,6.599,179.7323,-0.0880,0.0000
C00698=36.409,-119.516,6.598,179.0332,-0.2787,0.0000
C00699=33.027,-120.427,6.597,177.9550,-0.5107,0.0000
C00700=30.290,-121.060,6.595,176.5889,-0.7201,0.0000
C00701=28.099,-121.490,6.590,174.9904,-0.9229,0.0000
C00702=25.933,-121.876,6.584,173.3969,-1.1521,0.0000
C00703=23.250,-122.335,6.578,172.0415,-1.3416,0.0000
C00704=19.352,-122.957,6.573,171.1043,-1.3408,0.0000
C00705=13.651,-123.699,6.570,170.7093,-1.0235,0.0000
C00706=7.190,-124.241,6.570,170.6509,-0.5483,0.0000
C00707=0.000,-124.449,6.570,170.6405,0.0000,0.0000
C00708=0.000,-124.449,6.570,170.6405,0.0000,0.0000
C00709=-7.190,-124.241,6.570,170.6509,0.5483,0.0000
C00710=-13.651,-123.699,6.570,170.7093,1.0235,0.0000
C00711=-19.352,-122.957,6.573,171.1043,1.3408,0.0000
C00712=-23.250,-122.335,6.578,172.0415,1.3416,0.0000
C00713=-25.933,-121.876,6.584,173.3969,1.1521,0.0000
C00714=-28.099,-121.490,6.590,174.9904,0.9229,0.0000
C00715=-30.290,-121.060,6.595,176.5889,0.7201,0.0000
C00716=-33.027,-120.427,6.597,177.9550,0.5107,0.0000
C00717=-36.409,-119.516,6.598,179.0332,0.2787,0.0000
C00718=-39.998,-118.409,6.599,179.7323,0.0880,0.0000
C00719=-43.349,-117.240,6.599,179.9569,0.0159,0.0000
C00720=-46.376,-116.078,6.600,179.9949,0.0020,0.0000
C00721=-49.287,-114.873,6.600,179.9950,0.0021,0.0000
C00722=-52.249,-113.553,6.599,179.9583,0.0192,0.0000
C00723=-55.445,-112.011,6.599,179.7485,0.1271,0.0000
C00724=-58.765,-110.256,6.598,179.1193,0.4866,0.0000
C00725=-61.801,-108.508,6.597,178.1928,1.0854,0.0000
C00726=-64.184,-107.020,6.595,177.0785,1.9049,0.0000
C00727=-66.037,-105.776,6.590,175.8035,2.8963,0.0000
C00728=-67.842,-104.516,6.584,174.5122,3.8692,0.0000
C00729=-70.064,-102.945,6.578,173.4163,4.7046,0.0000
C00730=-73.260,-100.628,6.573,172.7494,5.3772,0.0000
C00731=-77.816,-97.121,6.570,172.6884,5.8831,0.0000
C00732=-82.768,-92.936,6.570,172.9775,6.2574,0.0000
C00733=-87.999,-87.999,6.570,173.3523,6.6477,0.0000
C00734=-92.936,-82.768,6.570,173.7426,7.0224,0.0000
C00735=-97.121,-77.816,6.570,174.1168,7.3116,0.0000
C00736=-100.628,-73.260,6.573,174.6229,7.2506,0.0000
C00737=-102.945,-70.064,6.578,175.2954,6.5837,0.0000
C00738=-104.516,-67.842,6.584,176.1308,5.4878,0.0000
C00739=-105.776,-66.037,6.590,177.1037,4.1965,0.0000
C00740=-107.020,-64.184,6.595,178.0951,2.9215,0.0000
C00741=-108.508,-61.801,6.597,178.9146,1.8072,0.0000
C00742=-110.256,-58.765,6.598,179.5134,0.8807,0.0000
C00743=-112.011,-55.445,6.599,179.8729,0.2515,0.0000
C00744=-113.553,-52.249,6.599,179.9808,0.0417,0.0000
C00745=-114.873,-49.287,6.600,179.9979,0.0050,0.0000
C00746=-116.078,-46.376,6.600,179.9980,0.0051,0.0000
C00747=-117.240,-43.349,6.599,179.9841,0.0431,0.0000
C00748=-118.409,-39.998,6.599,179.9120,0.2677,0.0000
C00749=-119.516,-36.409,6.598,179.7213,0.9668,0.0000
C00750=-120.427,-33.027,6.597,179.4893,2.0450,0.0000
C00751=-121.060,-30.290,6.595,179.2799,3.4111,0.0000
C00752=-121.490,-28.099,6.590,179.0771,5.0096,0.0000
C00753=-121.876,-25.933,6.584,178.8479,6.6031,0.0000
C00754=-122.335,-23.250,6.578,178.6584,7.9585,0.0000
C00755=-122.957,-19.352,6.573,178.6592,8.8957,0.0000
C00756=-123.699,-13.651,6.570,178.9765,9.2907,0.0000
C00757=-124.241,-7.190,6.570,179.4517,9.3491,0.0000
C00758=-124.449,0.000,6.570,-180.0000,9.3595,0.0000
C00759=-124.241,7.190,6.570,-179.4517,9.3491,0.0000
C00760=-123.699,13.651,6.570,-178.9765,9.2907,0.0000
C00761=-122.957,19.352,6.573,-178.6592,8.8957,0.0000
C00762=-122.335,23.250,6.578,-178.6584,7.9585,0.0000
C00763=-121.876,25.933,6.584,-178.8479,6.6031,0.0000
C00764=-121.490,28.099,6.590,-179.0771,5.0096,0.0000
C00765=-121.060,30.290,6.595,-179.2799,3.4111,0.0000
C00766=-120.427,33.027,6.597,-179.4893,2.0450,0.0000
C00767=-119.516,36.409,6.598,-179.7213,0.9668,0.0000
C00768=-118.409,39.998,6.599,-179.9120,0.2677,0.0000
C00769=-117.240,43.349,6.599,-179.9841,0.0431,0.0000
C00770=-116.078,46.376,6.600,-179.9980,0.0051,0.0000
C00771=-114.873,49.287,6.600,-179.9979,0.0050,0.0000
C00772=-113.553,52.249,6.599,-179.9808,0.0417,0.0000
C00773=-112.011,55.445,6.599,-179.8729,0.2515,0.0000
C00774=-110.256,58.765,6.598,-179.5134,0.8807,0.0000
C00775=-108.508,61.801,6.597,-178.9146,1.8072,0.0000
C00776=-107.020,64.184,6.595,-178.0951,2.9215,0.0000
C00777=-105.776,66.037,6.590,-177.1037,4.1965,0.0000
C00778=-104.516,67.842,6.584,-176.1308,5.4878,0.0000
C00779=-102.945,70.064,6.578,-175.2954,6.5837,0.0000
C00780=-100.628,73.260,6.573,-174.6228,7.2506,0.0000
C00781=-97.121,77.816,6.570,-174.1169,7.3116,0.0000
C00782=-92.936,82.768,6.570,-173.7426,7.0225,0.0000
C00783=-87.999,87.999,6.570,-173.3523,6.6477,0.0000
C00784=-82.768,92.936,6.570,-172.9776,6.2574,0.0000
C00785=-77.816,97.121,6.570,-172.6884,5.8832,0.0000
C00786=-73.260,100.628,6.573,-172.7494,5.3771,0.0000
C00787=-70.064,102.945,6.578,-173.4163,4.7046,0.0000
C00788=-67.842,104.516,6.584,-174.5122,3.8692,0.0000
C00789=-66.037,105.776,6.590,-175.8035,2.8963,0.0000
C00790=-64.184,107.020,6.595,-177.0785,1.9049,0.0000
C00791=-61.801,108.508,6.597,-178.1928,1.0854,0.0000
C00792=-58.765,110.256,6.598,-179.1193,0.4866,0.0000
C00793=-55.445,112.011,6.599,-179.7485,0.1271,0.0000
C00794=-52.249,113.553,6.599,-179.9583,0.0192,0.0000
C00795=-49.287,114.873,6.600,-179.9950,0.0021,0.0000
C00796=-46.376,116.078,6.600,-179.9949,0.0020,0.0000
C00797=-43.349,117.240,6.599,-179.9569,0.0159,0.0000
C00798=-39.998,118.409,6.599,-179.7323,0.0880,0.0000
C00799=-36.409,119.516,6.598,-179.0332,0.2787,0.0000
C00800=-33.027,120.427,6.597,-177.9550,0.5107,0.0000
C00801=-30.290,121.060,6.595,-176.5889,0.7201,0.0000
C00802=-28.099,121.490,6.590,-174.9904,0.9229,0.0000
C00803=-25.933,121.876,6.584,-173.3969,1.1521,0.0000
C00804=-23.250,122.335,6.578,-172.0415,1.3416,0.0000
C00805=-19.352,122.957,6.573,-171.1043,1.3408,0.0000
C00806=-13.651,123.699,6.570,-170.7093,1.0235,0.0000
C00807=-7.190,124.241,6.570,-170.6509,0.5483,0.0000
C00808=0.000,124.449,6.570,-170.6405,0.0000,0.0000
C00809=0.000,124.038,8.732,-167.8485,0.0000,0.0000
C00810=7.152,123.831,8.732,-167.8618,-0.7157,0.0000
C00811=13.588,123.293,8.732,-167.9360,-1.3249,0.0000
C00812=19.275,122.569,8.737,-168.4366,-1.6816,0.0000
C00813=23.159,121.990,8.749,-169.6379,-1.5733,0.0000
C00814=25.831,121.593,8.764,-171.4049,-1.2455,0.0000
C00815=27.992,121.281,8.778,-173.4987,-0.9622,0.0000
C00816=30.178,120.926,8.788,-175.5907,-0.7974,0.0000
C00817=32.905,120.361,8.792,-177.3695,-0.6059,0.0000
C00818=36.296,119.502,8.795,-178.7682,-0.3390,0.0000
C00819=39.909,118.425,8.797,-179.6664,-0.1072,0.0000
C00820=43.292,117.258,8.799,-179.9456,-0.0200,0.0000
C00821=46.357,116.086,8.800,-179.9937,-0.0025,0.0000
C00822=49.306,114.864,8.800,-179.9937,-0.0027,0.0000
C00823=52.302,113.527,8.799,-179.9474,-0.0243,0.0000
C00824=55.520,111.959,8.797,-179.6883,-0.1601,0.0000
C00825=58.836,110.166,8.795,-178.8893,-0.6314,0.0000
C00826=61.840,108.375,8.792,-177.7114,-1.4326,0.0000
C00827=64.169,106.846,8.788,-176.3172,-2.5584,0.0000
C00828=65.965,105.552,8.778,-174.7177,-3.9303,0.0000
C00829=67.714,104.245,8.764,-173.0301,-5.2283,0.0000
C00830=69.884,102.636,8.749,-171.5412,-6.2701,0.0000
C00831=73.040,100.299,8.737,-170.6062,-7.0640,0.0000
C00832=77.573,96.789,8.732,-170.4923,-7.6756,0.0000
C00833=82.504,92.619,8.732,-170.8586,-8.1522,0.0000
C00834=87.708,87.708,8.732,-171.3429,-8.6571,0.0000
C00835=92.619,82.504,8.732,-171.8478,-9.1414,0.0000
C00836=96.789,77.573,8.732,-172.3244,-9.5077,0.0000
C00837=100.299,73.040,8.737,-172.9360,-9.3937,0.0000
C00838=102.636,69.884,8.749,-173.7299,-8.4588,0.0000
C00839=104.245,67.714,8.764,-174.7717,-6.9699,0.0000
C00840=105.552,65.965,8.778,-176.0697,-5.2823,0.0000
C00841=106.846,64.169,8.788,-177.4416,-3.6828,0.0000
C00842=108.375,61.840,8.792,-178.5674,-2.2886,0.0000
C00843=110.166,58.836,8.795,-179.3686,-1.1107,0.0000
C00844=111.959,55.520,8.797,-179.8399,-0.3117,0.0000
C00845=113.527,52.302,8.799,-179.9757,-0.0526,0.0000
C00846=114.864,49.306,8.800,-179.9973,-0.0063,0.0000
C00847=116.086,46.357,8.800,-179.9975,-0.0063,0.0000
C00848=117.258,43.292,8.799,-179.9800,-0.0544,0.0000
C00849=118.425,39.909,8.797,-179.8928,-0.3336,0.0000
C00850=119.502,36.296,8.795,-179.6610,-1.2318,0.0000
C00851=120.361,32.905,8.792,-179.3941,-2.6305,0.0000
C00852=120.926,30.178,8.788,-179.2026,-4.4093,0.0000
C00853=121.281,27.992,8.778,-179.0378,-6.5013,0.0000
C00854=121.593,25.831,8.764,-178.7545,-8.5951,0.0000
C00855=121.990,23.159,8.749,-178.4267,-10.3621,0.0000
C00856=122.569,19.275,8.737,-178.3184,-11.5634,0.0000
C00857=123.293,13.588,8.732,-178.6751,-12.0640,0.0000
C00858=123.831,7.152,8.732,-179.2843,-12.1382,0.0000
C00859=124.038,0.000,8.732,180.0000,-12.1515,0.0000
C00860=123.831,-7.152,8.732,179.2844,-12.1381,0.0000
C00861=123.293,-13.588,8.732,178.6751,-12.0640,0.0000
C00862=122.569,-19.275,8.737,178.3184,-11.5634,0.0000
C00863=121.990,-23.159,8.749,178.4267,-10.3621,0.0000
C00864=121.593,-25.831,8.764,178.7545,-8.5951,0.0000
C00865=121.281,-27.992,8.778,179.0378,-6.5013,0.0000
C00866=120.926,-30.178,8.788,179.2026,-4.4093,0.0000
C00867=120.361,-32.905,8.792,179.3941,-2.6305,0.0000
C00868=119.502,-36.296,8.795,179.6610,-1.2318,0.0000
C00869=118.425,-39.909,8.797,179.8928,-0.3336,0.0000
C00870=117.258,-43.292,8.799,179.9800,-0.0544,0.0000
C00871=116.086,-46.357,8.800,179.9975,-0.0063,0.0000
C00872=114.864,-49.306,8.800,179.9973,-0.0063,0.0000
C00873=113.527,-52.302,8.799,179.9757,-0.0526,0.0000
C00874=111.959,-55.520,8.797,179.8399,-0.3117,0.0000
C00875=110.166,-58.836,8.795,179.3686,-1.1107,0.0000
C00876=108.375,-61.840,8.792,178.5674,-2.2886,0.0000
C00877=106.846,-64.169,8.788,177.4416,-3.6828,0.0000
C00878=105.552,-65.965,8.778,176.0697,-5.2823,0.0000
C00879=104.245,-67.714,8.764,174.7717,-6.9699,0.0000
C00880=102.636,-69.884,8.749,173.7299,-8.4588,0.0000
C00881=100.299,-73.040,8.737,172.9360,-9.3938,0.0000
C00882=96.789,-77.573,8.732,172.3244,-9.5077,0.0000
C00883=92.619,-82.504,8.732,171.8478,-9.1414,0.0000
C00884=87.708,-87.708,8.732,171.3429,-8.6571,0.0000
C00885=82.504,-92.619,8.732,170.8586,-8.1522,0.0000
C00886=77.573,-96.789,8.732,170.4923,-7.6756,0.0000
C00887=73.040,-100.299,8.737,170.6063,-7.0640,0.0000
C00888=69.884,-102.636,8.749,171.5412,-6.2701,0.0000
C00889=67.714,-104.245,8.764,173.0301,-5.2283,0.0000
C00890=65.965,-105.552,8.778,174.7177,-3.9303,0.0000
C00891=64.169,-106.846,8.788,176.3172,-2.5584,0.0000
C00892=61.840,-108.375,8.792,177.7114,-1.4326,0.0000
C00893=58.836,-110.166,8.795,178.8893,-0.6314,0.0000
C00894=55.520,-111.959,8.797,179.6883,-0.1601,0.0000
C00895=52.302,-113.527,8.799,179.9474,-0.0243,0.0000
C00896=49.306,-114.864,8.800,179.9937,-0.0027,0.0000
C00897=46.357,-116.086,8.800,179.9937,-0.0025,0.0000
C00898=43.292,-117.258,8.799,179.9456,-0.0200,0.0000
C00899=39.909,-118.425,8.797,179.6664,-0.1072,0.0000
C00900=36.296,-119.502,8.795,178.7682,-0.3390,0.0000
C00901=32.905,-120.361,8.792,177.3695,-0.6059,0.0000
C00902=30.178,-120.926,8.788,175.5907,-0.7974,0.0000
C00903=27.992,-121.281,8.778,173.4987,-0.9622,0.0000
C00904=25.831,-121.593,8.764,171.4049,-1.2455,0.0000
C00905=23.159,-121.990,8.749,169.6379,-1.5733,0.0000
C00906=19.275,-122.569,8.737,168.4366,-1.6816,0.0000
C00907=13.588,-123.293,8.732,167.9360,-1.3249,0.0000
C00908=7.152,-123.831,8.732,167.8618,-0.7157,0.0000
C00909=0.000,-124.038,8.732,167.8485,0.0000,0.0000
C00910=0.000,-124.038,8.732,167.8485,0.0000,0.0000
C00911=-7.152,-123.831,8.732,167.8619,0.7156,0.0000
C00912=-13.588,-123.293,8.732,167.9360,1.3249,0.0000
C00913=-19.275,-122.569,8.737,168.4366,1.6816,0.0000
C00914=-23.159,-121.990,8.749,169.6379,1.5733,0.0000
C00915=-25.831,-121.593,8.764,171.4049,1.2455,0.0000
C00916=-27.992,-121.281,8.778,173.4987,0.9622,0.0000
C00917=-30.178,-120.926,8.788,175.5907,0.7974,0.0000
C00918=-32.905,-120.361,8.792,177.3695,0.6059,0.0000
C00919=-36.296,-119.502,8.795,178.7682,0.3390,0.0000
C00920=-39.909,-118.425,8.797,179.6664,0.1072,0.0000
C00921=-43.292,-117.258,8.799,179.9456,0.0200,0.0000
C00922=-46.357,-116.086,8.800,179.9937,0.0025,0.0000
C00923=-49.306,-114.864,8.800,179.9937,0.0027,0.0000
C00924=-52.302,-113.527,8.799,179.9474,0.0243,0.0000
C00925=-55.520,-111.959,8.797,179.6883,0.1601,0.0000
C00926=-58.836,-110.166,8.795,178.8893,0.6314,0.0000
C00927=-61.840,-108.375,8.792,177.7114,1.4326,0.0000
C00928=-64.169,-106.846,8.788,176.3172,2.5584,0.0000
C00929=-65.965,-105.552,8.778,174.7177,3.9303,0.0000
C00930=-67.714,-104.245,8.764,173.0301,5.2283,0.0000
C00931=-69.884,-102.636,8.749,171.5412,6.2701,0.0000
C00932=-73.040,-100.299,8.737,170.6062,7.0640,0.0000
C00933=-77.573,-96.789,8.732,170.4923,7.6756,0.0000
C00934=-82.504,-92.619,8.732,170.8586,8.1522,0.0000
C00935=-87.708,-87.708,8.732,171.3429,8.6571,0.0000
C00936=-92.619,-82.504,8.732,171.8478,9.1414,0.0000
C00937=-96.789,-77.573,8.732,172.3244,9.5077,0.0000
C00938=-100.299,-73.040,8.737,172.9360,9.3937,0.0000
C00939=-102.636,-69.884,8.749,173.7299,8.4588,0.0000
C00940=-104.245,-67.714,8.764,174.7717,6.9699,0.0000
C00941=-105.552,-65.965,8.778,176.0697,5.2823,0.0000
C00942=-106.846,-64.169,8.788,177.4416,3.6828,0.0000
C00943=-108.375,-61.840,8.792,178.5674,2.2886,0.0000
C00944=-110.166,-58.836,8.795,179.3686,1.1107,0.0000
C00945=-111.959,-55.520,8.797,179.8399,0.3117,0.0000
C00946=-113.527,-52.302,8.799,179.9757,0.0526,0.0000
C00947=-114.864,-49.306,8.800,179.9973,0.0063,0.0000
C00948=-116.086,-46.357,8.800,179.9975,0.0063,0.0000
C00949=-117.258,-43.292,8.799,179.9800,0.0544,0.0000
C00950=-118.425,-39.909,8.797,179.8928,0.3336,0.0000
C00951=-119.502,-36.296,8.795,179.6610,1.2318,0.0000
C00952=-120.361,-32.905,8.792,179.3941,2.6305,0.0000
C00953=-120.926,-30.178,8.788,179.2026,4.4093,0.0000
C00954=-121.281,-27.992,8.778,179.0378,6.5013,0.0000
C00955=-121.593,-25.831,8.764,178.7545,8.5951,0.0000
C00956=-121.990,-23.159,8.749,178.4267,10.3621,0.0000
C00957=-122.569,-19.275,8.737,178.3184,11.5634,0.0000
C00958=-123.293,-13.588,8.732,178.6751,12.0640,0.0000
C00959=-123.831,-7.152,8.732,179.2843,12.1382,0.0000
C00960=-124.038,0.000,8.732,-180.0000,12.1515,0.0000
C00961=-123.831,7.152,8.732,-179.2844,12.1381,0.0000
C00962=-123.293,13.588,8.732,-178.6751,12.0640,0.0000
C00963=-122.569,19.275,8.737,-178.3184,11.5634,0.0000
C00964=-121.990,23.159,8.749,-178.4267,10.3621,0.0000
C00965=-121.593,25.831,8.764,-178.7545,8.5951,0.0000
C00966=-121.281,27.992,8.778,-179.0378,6.5013,0.0000
C00967=-120.926,30.178,8.788,-179.2026,4.4093,0.0000
C00968=-120.361,32.905,8.792,-179.3941,2.6305,0.0000
C00969=-119.502,36.296,8.795,-179.6610,1.2318,0.0000
C00970=-118.425,39.909,8.797,-179.8928,0.3336,0.0000
C00971=-117.258,43.292,8.799,-179.9800,0.0544,0.0000
C00972=-116.086,46.357,8.800,-179.9975,0.0063,0.0000
C00973=-114.864,49.306,8.800,-179.9973,0.0063,0.0000
C00974=-113.527,52.302,8.799,-179.9757,0.0526,0.0000
C00975=-111.959,55.520,8.797,-179.8399,0.3117,0.0000
C00976=-110.166,58.836,8.795,-179.3686,1.1107,0.0000
C00977=-108.375,61.840,8.792,-178.5674,2.2886,0.0000
C00978=-106.846,64.169,8.788,-177.4416,3.6828,0.0000
C00979=-105.552,65.965,8.778,-176.0697,5.2823,0.0000
C00980=-104.245,67.714,8.764,-174.7717,6.9699,0.0000
C00981=-102.636,69.884,8.749,-173.7299,8.4588,0.0000
C00982=-100.299,73.040,8.737,-172.9360,9.3938,0.0000
C00983=-96.789,77.573,8.732,-172.3244,9.5077,0.0000
C00984=-92.619,82.504,8.732,-171.8478,9.1414,0.0000
C00985=-87.708,87.708,8.732,-171.3429,8.6571,0.0000
C00986=-82.504,92.619,8.732,-170.8586,8.1522,0.0000
C00987=-77.573,96.789,8.732,-170.4923,7.6756,0.0000
C00988=-73.040,100.299,8.737,-170.6063,7.0640,0.0000
C00989=-69.884,102.636,8.749,-171.5412,6.2701,0.0000
C00990=-67.714,104.245,8.764,-173.0301,5.2283,0.0000
C00991=-65.965,105.552,8.778,-174.7177,3.9303,0.0000
C00992=-64.169,106.846,8.788,-176.3172,2.5584,0.0000
C00993=-61.840,108.375,8.792,-177.7114,1.4326,0.0000
C00994=-58.836,110.166,8.795,-178.8893,0.6314,0.0000
C00995=-55.520,111.959,8.797,-179.6883,0.1601,0.0000
C00996=-52.302,113.527,8.799,-179.9474,0.0243,0.0000
C00997=-49.306,114.864,8.800,-179.9937,0.0027,0.0000
C00998=-46.357,116.086,8.800,-179.9937,0.0025,0.0000
C00999=-43.292,117.258,8.799,-179.9456,0.0200,0.0000
C01000=-39.909,118.425,8.797,-179.6664,0.1072,0.0000
C01001=-36.296,119.502,8.795,-178.7682,0.3390,0.0000
C01002=-32.905,120.361,8.792,-177.3695,0.6059,0.0000
C01003=-30.178,120.926,8.788,-175.5907,0.7974,0.0000
C01004=-27.992,121.281,8.778,-173.4987,0.9622,0.0000
C01005=-25.831,121.593,8.764,-171.4049,1.2455,0.0000
C01006=-23.159,121.990,8.749,-169.6379,1.5733,0.0000
C01007=-19.275,122.569,8.737,-168.4366,1.6816,0.0000
C01008=-13.588,123.293,8.732,-167.9360,1.3249,0.0000
C01009=-7.152,123.831,8.732,-167.8619,0.7156,0.0000
C01010=0.000,124.038,8.732,-167.8485,0.0000,0.0000
C01011=0.000,123.526,10.871,-165.2403,0.0000,0.0000
C01012=7.105,123.320,10.871,-165.2564,-0.8746,0.0000
C01013=13.509,122.787,10.871,-165.3441,-1.6024,0.0000
C01014=19.180,122.085,10.881,-165.9353,-1.9495,0.0000
C01015=23.045,121.559,10.903,-167.3801,-1.6455,0.0000
C01016=25.704,121.239,10.931,-169.5534,-1.1205,0.0000
C01017=27.858,121.018,10.958,-172.1395,-0.8022,0.0000
C01018=30.036,120.757,10.977,-174.6912,-0.7561,0.0000
C01019=32.753,120.278,10.986,-176.8486,-0.6486,0.0000
C01020=36.153,119.485,10.990,-178.5415,-0.3776,0.0000
C01021=39.796,118.446,10.994,-179.6165,-0.1196,0.0000
C01022=43.221,117.282,10.997,-179.9364,-0.0233,0.0000
C01023=46.333,116.095,11.000,-179.9926,-0.0029,0.0000
C01024=49.329,114.854,11.000,-179.9927,-0.0031,0.0000
C01025=52.369,113.493,10.997,-179.9386,-0.0286,0.0000
C01026=55.614,111.894,10.994,-179.6442,-0.1866,0.0000
C01027=58.925,110.053,10.990,-178.7017,-0.7645,0.0000
C01028=61.889,108.209,10.986,-177.3127,-1.7714,0.0000
C01029=64.150,106.627,10.977,-175.7087,-3.2266,0.0000
C01030=65.874,105.271,10.958,-173.8630,-5.0132,0.0000
C01031=67.554,103.905,10.931,-171.7943,-6.6474,0.0000
C01032=69.660,102.250,10.903,-169.8722,-7.8573,0.0000
C01033=72.765,99.889,10.881,-168.6229,-8.7033,0.0000
C01034=77.271,96.376,10.871,-168.4311,-9.3774,0.0000
C01035=82.176,92.225,10.871,-168.8623,-9.9422,0.0000
C01036=87.346,87.346,10.871,-169.4472,-10.5529,0.0000
C01037=92.225,82.176,10.871,-170.0578,-11.1377,0.0000
C01038=96.376,77.271,10.871,-170.6225,-11.5689,0.0000
C01039=99.889,72.765,10.881,-171.2967,-11.3771,0.0000
C01040=102.250,69.660,10.903,-172.1427,-10.1278,0.0000
C01041=103.905,67.554,10.931,-173.3526,-8.2057,0.0000
C01042=105.271,65.874,10.958,-174.9868,-6.1370,0.0000
C01043=106.627,64.150,10.977,-176.7734,-4.2913,0.0000
C01044=108.209,61.889,10.986,-178.2286,-2.6873,0.0000
C01045=110.053,58.925,10.990,-179.2355,-1.2983,0.0000
C01046=111.894,55.614,10.994,-179.8134,-0.3558,0.0000
C01047=113.493,52.369,10.997,-179.9714,-0.0614,0.0000
C01048=114.854,49.329,11.000,-179.9969,-0.0073,0.0000
C01049=116.095,46.333,11.000,-179.9971,-0.0074,0.0000
C01050=117.282,43.221,10.997,-179.9767,-0.0636,0.0000
C01051=118.446,39.796,10.994,-179.8804,-0.3835,0.0000
C01052=119.485,36.153,10.990,-179.6224,-1.4585,0.0000
C01053=120.278,32.753,10.986,-179.3514,-3.1514,0.0000
C01054=120.757,30.036,10.977,-179.2439,-5.3088,0.0000
C01055=121.018,27.858,10.958,-179.1978,-7.8605,0.0000
C01056=121.239,25.704,10.931,-178.8795,-10.4466,0.0000
C01057=121.559,23.045,10.903,-178.3545,-12.6199,0.0000
C01058=122.085,19.180,10.881,-178.0505,-14.0647,0.0000
C01059=122.787,13.509,10.871,-178.3976,-14.6559,0.0000
C01060=123.320,7.105,10.871,-179.1254,-14.7436,0.0000
C01061=123.526,0.000,10.871,180.0000,-14.7597,0.0000
C01062=123.320,-7.105,10.871,179.1255,-14.7436,0.0000
C01063=122.787,-13.509,10.871,178.3977,-14.6560,0.0000
C01064=122.085,-19.180,10.881,178.0504,-14.0647,0.0000
C01065=121.559,-23.045,10.903,178.3545,-12.6199,0.0000
C01066=121.239,-25.704,10.931,178.8795,-10.4466,0.0000
C01067=121.018,-27.858,10.958,179.1978,-7.8605,0.0000
C01068=120.757,-30.036,10.977,179.2439,-5.3088,0.0000
C01069=120.278,-32.753,10.986,179.3514,-3.1514,0.0000
C01070=119.485,-36.153,10.990,179.6224,-1.4585,0.0000
C01071=118.446,-39.796,10.994,179.8804,-0.3835,0.0000
C01072=117.282,-43.221,10.997,179.9767,-0.0636,0.0000
C01073=116.095,-46.333,11.000,179.9971,-0.0074,0.0000
C01074=114.854,-49.329,11.000,179.9969,-0.0073,0.0000
C01075=113.493,-52.369,10.997,179.9714,-0.0614,0.0000
C01076=111.894,-55.614,10.994,179.8134,-0.3558,0.0000
C01077=110.053,-58.925,10.990,179.2355,-1.2983,0.0000
C01078=108.209,-61.889,10.986,178.2286,-2.6873,0.0000
C01079=106.627,-64.150,10.977,176.7734,-4.2913,0.0000
C01080=105.271,-65.874,10.958,174.9868,-6.1370,0.0000
C01081=103.905,-67.554,10.931,173.3526,-8.2057,0.0000
C01082=102.250,-69.660,10.903,172.1427,-10.1278,0.0000
C01083=99.889,-72.765,10.881,171.2967,-11.3771,0.0000
C01084=96.376,-77.271,10.871,170.6226,-11.5689,0.0000
C01085=92.225,-82.176,10.871,170.0578,-11.1377,0.0000
C01086=87.346,-87.346,10.871,169.4471,-10.5528,0.0000
C01087=82.176,-92.225,10.871,168.8623,-9.9422,0.0000
C01088=77.271,-96.376,10.871,168.4311,-9.3775,0.0000
C01089=72.765,-99.889,10.881,168.6229,-8.7033,0.0000
C01090=69.660,-102.250,10.903,169.8722,-7.8573,0.0000
C01091=67.554,-103.905,10.931,171.7943,-6.6474,0.0000
C01092=65.874,-105.271,10.958,173.8630,-5.0132,0.0000
C01093=64.150,-106.627,10.977,175.7087,-3.2266,0.0000
C01094=61.889,-108.209,10.986,177.3127,-1.7714,0.0000
C01095=58.925,-110.053,10.990,178.7017,-0.7645,0.0000
C01096=55.614,-111.894,10.994,179.6442,-0.1866,0.0000
C01097=52.369,-113.493,10.997,179.9386,-0.0286,0.0000
C01098=49.329,-114.854,11.000,179.9927,-0.0031,0.0000
C01099=46.333,-116.095,11.000,179.9926,-0.0029,0.0000
C01100=43.221,-117.282,10.997,179.9364,-0.0233,0.0000
C01101=39.796,-118.446,10.994,179.6165,-0.1196,0.0000
C01102=36.153,-119.485,10.990,178.5415,-0.3776,0.0000
C01103=32.753,-120.278,10.986,176.8486,-0.6486,0.0000
C01104=30.036,-120.757,10.977,174.6912,-0.7561,0.0000
C01105=27.858,-121.018,10.958,172.1395,-0.8022,0.0000
C01106=25.704,-121.239,10.931,169.5534,-1.1205,0.0000
C01107=23.045,-121.559,10.903,167.3801,-1.6455,0.0000
C01108=19.180,-122.085,10.881,165.9353,-1.9495,0.0000
C01109=13.509,-122.787,10.871,165.3441,-1.6024,0.0000
C01110=7.105,-123.320,10.871,165.2564,-0.8746,0.0000
C01111=0.000,-123.526,10.871,165.2403,0.0000,0.0000
C01112=0.000,-123.526,10.871,165.2403,0.0000,0.0000
C01113=-7.105,-123.320,10.871,165.2564,0.8745,0.0000
C01114=-13.509,-122.787,10.871,165.3440,1.6023,0.0000
C01115=-19.180,-122.085,10.881,165.9353,1.9496,0.0000
C01116=-23.045,-121.559,10.903,167.3801,1.6455,0.0000
C01117=-25.704,-121.239,10.931,169.5534,1.1205,0.0000
C01118=-27.858,-121.018,10.958,172.1395,0.8022,0.0000
C01119=-30.036,-120.757,10.977,174.6912,0.7561,0.0000
C01120=-32.753,-120.278,10.986,176.8486,0.6486,0.0000
C01121=-36.153,-119.485,10.990,178.5415,0.3776,0.0000
C01122=-39.796,-118.446,10.994,179.6165,0.1196,0.0000
C01123=-43.221,-117.282,10.997,179.9364,0.0233,0.0000
C01124=-46.333,-116.095,11.000,179.9926,0.0029,0.0000
C01125=-49.329,-114.854,11.000,179.9927,0.0031,0.0000
C01126=-52.369,-113.493,10.997,179.9386,0.0286,0.0000
C01127=-55.614,-111.894,10.994,179.6442,0.1866,0.0000
C01128=-58.925,-110.053,10.990,178.7017,0.7645,0.0000
C01129=-61.889,-108.209,10.986,177.3127,1.7714,0.0000
C01130=-64.150,-106.627,10.977,175.7087,3.2266,0.0000
C01131=-65.874,-105.271,10.958,173.8630,5.0132,0.0000
C01132=-67.554,-103.905,10.931,171.7943,6.6474,0.0000
C01133=-69.660,-102.250,10.903,169.8722,7.8573,0.0000
C01134=-72.765,-99.889,10.881,168.6229,8.7033,0.0000
C01135=-77.271,-96.376,10.871,168.4311,9.3774,0.0000
C01136=-82.176,-92.225,10.871,168.8623,9.9422,0.0000
C01137=-87.346,-87.346,10.871,169.4472,10.5529,0.0000
C01138=-92.225,-82.176,10.871,170.0578,11.1377,0.0000
C01139=-96.376,-77.271,10.871,170.6225,11.5689,0.0000
C01140=-99.889,-72.765,10.881,171.2967,11.3771,0.0000
C01141=-102.250,-69.660,10.903,172.1427,10.1278,0.0000
C01142=-103.905,-67.554,10.931,173.3526,8.2057,0.0000
C01143=-105.271,-65.874,10.958,174.9868,6.1370,0.0000
C01144=-106.627,-64.150,10.977,176.7734,4.2913,0.0000
C01145=-108.209,-61.889,10.986,178.2286,2.6873,0.0000
C01146=-110.053,-58.925,10.990,179.2355,1.2983,0.0000
C01147=-111.894,-55.614,10.994,179.8134,0.3558,0.0000
C01148=-113.493,-52.369,10.997,179.9714,0.0614,0.0000
C01149=-114.854,-49.329,11.000,179.9969,0.0073,0.0000
C01150=-116.095,-46.333,11.000,179.9971,0.0074,0.0000
C01151=-117.282,-43.221,10.997,179.9767,0.0636,0.0000
C01152=-118.446,-39.796,10.994,179.8804,0.3835,0.0000
C01153=-119.485,-36.153,10.990,179.6224,1.4585,0.0000
C01154=-120.278,-32.753,10.986,179.3514,3.1514,0.0000
C01155=-120.757,-30.036,10.977,179.2439,5.3088,0.0000
C01156=-121.018,-27.858,10.958,179.1978,7.8605,0.0000
C01157=-121.239,-25.704,10.931,178.8795,10.4466,0.0000
C01158=-121.559,-23.045,10.903,178.3545,12.6199,0.0000
C01159=-122.085,-19.180,10.881,178.0505,14.0647,0.0000
C01160=-122.787,-13.509,10.871,178.3976,14.6559,0.0000
C01161=-123.320,-7.105,10.871,179.1254,14.7436,0.0000
C01162=-123.526,0.000,10.871,-180.0000,14.7597,0.0000
C01163=-123.320,7.105,10.871,-179.1255,14.7436,0.0000
C01164=-122.787,13.509,10.871,-178.3977,14.6560,0.0000
C01165=-122.085,19.180,10.881,-178.0504,14.0647,0.0000
C01166=-121.559,23.045,10.903,-178.3545,12.6199,0.0000
C01167=-121.239,25.704,10.931,-178.8795,10.4466,0.0000
C01168=-121.018,27.858,10.958,-179.1978,7.8605,0.0000
C01169=-120.757,30.036,10.977,-179.2439,5.3088,0.0000
C01170=-120.278,32.753,10.986,-179.3514,3.1514,0.0000
C01171=-119.485,36.153,10.990,-179.6224,1.4585,0.0000
C01172=-118.446,39.796,10.994,-179.8804,0.3835,0.0000
C01173=-117.282,43.221,10.997,-179.9767,0.0636,0.0000
C01174=-116.095,46.333,11.000,-179.9971,0.0074,0.0000
C01175=-114.854,49.329,11.000,-179.9969,0.0073,0.0000
C01176=-113.493,52.369,10.997,-179.9714,0.0614,0.0000
C01177=-111.894,55.614,10.994,-179.8134,0.3558,0.0000
C01178=-110.053,58.925,10.990,-179.2355,1.2983,0.0000
C01179=-108.209,61.889,10.986,-178.2286,2.6873,0.0000
C01180=-106.627,64.150,10.977,-176.7734,4.2913,0.0000
C01181=-105.271,65.874,10.958,-174.9868,6.1370,0.0000
C01182=-103.905,67.554,10.931,-173.3526,8.2057,0.0000
C01183=-102.250,69.660,10.903,-172.1427,10.1278,0.0000
C01184=-99.889,72.765,10.881,-171.2967,11.3771,0.0000
C01185=-96.376,77.271,10.871,-170.6226,11.5689,0.0000
C01186=-92.225,82.176,10.871,-170.0578,11.1377,0.0000
C01187=-87.346,87.346,10.871,-169.4471,10.5528,0.0000
C01188=-82.176,92.225,10.871,-168.8623,9.9422,0.0000
C01189=-77.271,96.376,10.871,-168.4311,9.3775,0.0000
C01190=-72.765,99.889,10.881,-168.6229,8.7033,0.0000
C01191=-69.660,102.250,10.903,-169.8722,7.8573,0.0000
C01192=-67.554,103.905,10.931,-171.7943,6.6474,0.0000
C01193=-65.874,105.271,10.958,-173.8630,5.0132,0.0000
C01194=-64.150,106.627,10.977,-175.7087,3.2266,0.0000
C01195=-61.889,108.209,10.986,-177.3127,1.7714,0.0000
C01196=-58.925,110.053,10.990,-178.7017,0.7645,0.0000
C01197=-55.614,111.894,10.994,-179.6442,0.1866,0.0000
C01198=-52.369,113.493,10.997,-179.9386,0.0286,0.0000
C01199=-49.329,114.854,11.000,-179.9927,0.0031,0.0000
C01200=-46.333,116.095,11.000,-179.9926,0.0029,0.0000
C01201=-43.221,117.282,10.997,-179.9364,0.0233,0.0000
C01202=-39.796,118.446,10.994,-179.6165,0.1196,0.0000
C01203=-36.153,119.485,10.990,-178.5415,0.3776,0.0000
C01204=-32.753,120.278,10.986,-176.8486,0.6486,0.0000
C01205=-30.036,120.757,10.977,-174.6912,0.7561,0.0000
C01206=-27.858,121.018,10.958,-172.1395,0.8022,0.0000
C01207=-25.704,121.239,10.931,-169.5534,1.1205,0.0000
C01208=-23.045,121.559,10.903,-167.3801,1.6455,0.0000
C01209=-19.180,122.085,10.881,-165.9353,1.9496,0.0000
C01210=-13.509,122.787,10.871,-165.3440,1.6023,0.0000
C01211=-7.105,123.320,10.871,-165.2564,0.8745,0.0000
C01212=0.000,123.526,10.871,-165.2403,0.0000,0.0000
C01213=0.000,122.920,12.986,-162.8181,0.0001,0.0000
C01214=7.050,122.716,12.986,-162.8365,-1.0250,0.0000
C01215=13.416,122.189,12.986,-162.9355,-1.8543,0.0000
C01216=19.067,121.511,13.002,-163.6037,-2.1363,0.0000
C01217=22.909,121.048,13.039,-165.2824,-1.5339,0.0000
C01218=25.553,120.818,13.086,-167.8783,-0.7475,0.0000
C01219=27.698,120.705,13.130,-170.9569,-0.4216,0.0000
C01220=29.867,120.556,13.161,-173.9169,-0.5842,0.0000
C01221=32.570,120.178,13.176,-176.4033,-0.6343,0.0000
C01222=35.982,119.464,13.183,-178.3578,-0.3934,0.0000
C01223=39.661,118.471,13.189,-179.5843,-0.1252,0.0000
C01224=43.136,117.310,13.196,-179.9293,-0.0257,0.0000
C01225=46.304,116.106,13.199,-179.9918,-0.0032,0.0000
C01226=49.357,114.841,13.199,-179.9919,-0.0035,0.0000
C01227=52.449,113.453,13.196,-179.9318,-0.0318,0.0000
C01228=55.727,111.816,13.189,-179.6175,-0.2055,0.0000
C01229=59.031,109.917,13.183,-178.5606,-0.8832,0.0000
C01230=61.948,108.010,13.176,-177.0075,-2.0971,0.0000
C01231=64.127,106.365,13.161,-175.2800,-3.8985,0.0000
C01232=65.766,104.936,13.130,-173.2847,-6.1265,0.0000
C01233=67.363,103.500,13.086,-170.8485,-8.1182,0.0000
C01234=69.395,101.793,13.039,-168.4328,-9.4699,0.0000
C01235=72.439,99.404,13.002,-166.8059,-10.2975,0.0000
C01236=76.914,95.887,12.986,-166.5071,-10.9880,0.0000
C01237=81.788,91.759,12.986,-166.9905,-11.6259,0.0000
C01238=86.917,86.917,12.986,-167.6669,-12.3332,0.0000
C01239=91.759,81.788,12.986,-168.3740,-13.0094,0.0000
C01240=95.887,76.914,12.986,-169.0119,-13.4928,0.0000
C01241=99.404,72.439,13.002,-169.7026,-13.1941,0.0000
C01242=101.793,69.395,13.039,-170.5301,-11.5672,0.0000
C01243=103.500,67.363,13.086,-171.8818,-9.1515,0.0000
C01244=104.936,65.766,13.130,-173.8735,-6.7153,0.0000
C01245=106.365,64.127,13.161,-176.1015,-4.7200,0.0000
C01246=108.010,61.948,13.176,-177.9029,-2.9925,0.0000
C01247=109.917,59.031,13.183,-179.1168,-1.4394,0.0000
C01248=111.816,55.727,13.189,-179.7945,-0.3825,0.0000
C01249=113.453,52.449,13.196,-179.9682,-0.0682,0.0000
C01250=114.841,49.357,13.199,-179.9965,-0.0081,0.0000
C01251=116.106,46.304,13.199,-179.9968,-0.0082,0.0000
C01252=117.310,43.136,13.196,-179.9743,-0.0707,0.0000
C01253=118.471,39.661,13.189,-179.8748,-0.4157,0.0000
C01254=119.464,35.982,13.183,-179.6066,-1.6422,0.0000
C01255=120.178,32.570,13.176,-179.3657,-3.5967,0.0000
C01256=120.556,29.867,13.161,-179.4158,-6.0831,0.0000
C01257=120.705,27.698,13.130,-179.5784,-9.0431,0.0000
C01258=120.818,25.553,13.086,-179.2525,-12.1217,0.0000
C01259=121.048,22.909,13.039,-178.4661,-14.7176,0.0000
C01260=121.511,19.067,13.002,-177.8637,-16.3963,0.0000
C01261=122.189,13.416,12.986,-178.1457,-17.0645,0.0000
C01262=122.716,7.050,12.986,-178.9750,-17.1635,0.0000
C01263=122.920,0.000,12.986,179.9999,-17.1819,0.0000
C01264=122.716,-7.050,12.986,178.9751,-17.1635,0.0000
C01265=122.189,-13.416,12.986,178.1458,-17.0645,0.0000
C01266=121.511,-19.067,13.002,177.8637,-16.3962,0.0000
C01267=121.048,-22.909,13.039,178.4661,-14.7176,0.0000
C01268=120.818,-25.553,13.086,179.2525,-12.1217,0.0000
C01269=120.705,-27.698,13.130,179.5784,-9.0431,0.0000
C01270=120.556,-29.867,13.161,179.4158,-6.0831,0.0000
C01271=120.178,-32.570,13.176,179.3657,-3.5967,0.0000
C01272=119.464,-35.982,13.183,179.6066,-1.6422,0.0000
C01273=118.471,-39.661,13.189,179.8748,-0.4157,0.0000
C01274=117.310,-43.136,13.196,179.9743,-0.0707,0.0000
C01275=116.106,-46.304,13.199,179.9968,-0.0082,0.0000
C01276=114.841,-49.357,13.199,179.9965,-0.0081,0.0000
C01277=113.453,-52.449,13.196,179.9682,-0.0682,0.0000
C01278=111.816,-55.727,13.189,179.7945,-0.3825,0.0000
C01279=109.917,-59.031,13.183,179.1168,-1.4394,0.0000
C01280=108.010,-61.948,13.176,177.9029,-2.9925,0.0000
C01281=106.365,-64.127,13.161,176.1015,-4.7200,0.0000
C01282=104.936,-65.766,13.130,173.8735,-6.7153,0.0000
C01283=103.500,-67.363,13.086,171.8818,-9.1515,0.0000
C01284=101.793,-69.395,13.039,170.5301,-11.5672,0.0000
C01285=99.404,-72.439,13.002,169.7025,-13.1941,0.0000
C01286=95.887,-76.914,12.986,169.0120,-13.4929,0.0000
C01287=91.759,-81.788,12.986,168.3741,-13.0095,0.0000
C01288=86.917,-86.917,12.986,167.6668,-12.3331,0.0000
C01289=81.788,-91.759,12.986,166.9906,-11.6260,0.0000
C01290=76.914,-95.887,12.986,166.5072,-10.9881,0.0000
C01291=72.439,-99.404,13.002,166.8059,-10.2974,0.0000
C01292=69.395,-101.793,13.039,168.4328,-9.4699,0.0000
C01293=67.363,-103.500,13.086,170.8485,-8.1182,0.0000
C01294=65.766,-104.936,13.130,173.2847,-6.1265,0.0000
C01295=64.127,-106.365,13.161,175.2800,-3.8985,0.0000
C01296=61.948,-108.010,13.176,177.0075,-2.0971,0.0000
C01297=59.031,-109.917,13.183,178.5606,-0.8832,0.0000
C01298=55.727,-111.816,13.189,179.6175,-0.2055,0.0000
C01299=52.449,-113.453,13.196,179.9318,-0.0318,0.0000
C01300=49.357,-114.841,13.199,179.9919,-0.0035,0.0000
C01301=46.304,-116.106,13.199,179.9918,-0.0032,0.0000
C01302=43.136,-117.310,13.196,179.9293,-0.0257,0.0000
C01303=39.661,-118.471,13.189,179.5843,-0.1252,0.0000
C01304=35.982,-119.464,13.183,178.3578,-0.3934,0.0000
C01305=32.570,-120.178,13.176,176.4033,-0.6343,0.0000
C01306=29.867,-120.556,13.161,173.9169,-0.5842,0.0000
C01307=27.698,-120.705,13.130,170.9569,-0.4216,0.0000
C01308=25.553,-120.818,13.086,167.8783,-0.7475,0.0000
C01309=22.909,-121.048,13.039,165.2824,-1.5339,0.0000
C01310=19.067,-121.511,13.002,163.6037,-2.1363,0.0000
C01311=13.416,-122.189,12.986,162.9355,-1.8543,0.0000
C01312=7.050,-122.716,12.986,162.8365,-1.0250,0.0000
C01313=0.000,-122.920,12.986,162.8181,0.0001,0.0000
C01314=0.000,-122.920,12.986,162.8181,0.0001,0.0000
C01315=-7.050,-122.716,12.986,162.8365,1.0249,0.0000
C01316=-13.416,-122.189,12.986,162.9355,1.8542,0.0000
C01317=-19.067,-121.511,13.002,163.6038,2.1363,0.0000
C01318=-22.909,-121.048,13.039,165.2824,1.5339,0.0000
C01319=-25.553,-120.818,13.086,167.8783,0.7475,0.0000
C01320=-27.698,-120.705,13.130,170.9569,0.4216,0.0000
C01321=-29.867,-120.556,13.161,173.9169,0.5842,0.0000
C01322=-32.570,-120.178,13.176,176.4033,0.6343,0.0000
C01323=-35.982,-119.464,13.183,178.3578,0.3934,0.0000
C01324=-39.661,-118.471,13.189,179.5843,0.1252,0.0000
C01325=-43.136,-117.310,13.196,179.9293,0.0257,0.0000
C01326=-46.304,-116.106,13.199,179.9918,0.0032,0.0000
C01327=-49.357,-114.841,13.199,179.9919,0.0035,0.0000
C01328=-52.449,-113.453,13.196,179.9318,0.0318,0.0000
C01329=-55.727,-111.816,13.189,179.6175,0.2055,0.0000
C01330=-59.031,-109.917,13.183,178.5606,0.8832,0.0000
C01331=-61.948,-108.010,13.176,177.0075,2.0971,0.0000
C01332=-64.127,-106.365,13.161,175.2800,3.8985,0.0000
C01333=-65.766,-104.936,13.130,173.2847,6.1265,0.0000
C01334=-67.363,-103.500,13.086,170.8485,8.1182,0.0000
C01335=-69.395,-101.793,13.039,168.4328,9.4699,0.0000
C01336=-72.439,-99.404,13.002,166.8059,10.2975,0.0000
C01337=-76.914,-95.887,12.986,166.5071,10.9880,0.0000
C01338=-81.788,-91.759,12.986,166.9905,11.6259,0.0000
C01339=-86.917,-86.917,12.986,167.6669,12.3332,0.0000
C01340=-91.759,-81.788,12.986,168.3740,13.0094,0.0000
C01341=-95.887,-76.914,12.986,169.0119,13.4928,0.0000
C01342=-99.404,-72.439,13.002,169.7026,13.1941,0.0000
C01343=-101.793,-69.395,13.039,170.5301,11.5672,0.0000
C01344=-103.500,-67.363,13.086,171.8818,9.1515,0.0000
C01345=-104.936,-65.766,13.130,173.8735,6.7153,0.0000
C01346=-106.365,-64.127,13.161,176.1015,4.7200,0.0000
C01347=-108.010,-61.948,13.176,177.9029,2.9925,0.0000
C01348=-109.917,-59.031,13.183,179.1168,1.4394,0.0000
C01349=-111.816,-55.727,13.189,179.7945,0.3825,0.0000
C01350=-113.453,-52.449,13.196,179.9682,0.0682,0.0000
C01351=-114.841,-49.357,13.199,179.9965,0.0081,0.0000
C01352=-116.106,-46.304,13.199,179.9968,0.0082,0.0000
C01353=-117.310,-43.136,13.196,179.9743,0.0707,0.0000
C01354=-118.471,-39.661,13.189,179.8748,0.4157,0.0000
C01355=-119.464,-35.982,13.183,179.6066,1.6422,0.0000
C01356=-120.178,-32.570,13.176,179.3657,3.5967,0.0000
C01357=-120.556,-29.867,13.161,179.4158,6.0831,0.0000
C01358=-120.705,-27.698,13.130,179.5784,9.0431,0.0000
C01359=-120.818,-25.553,13.086,179.2525,12.1217,0.0000
C01360=-121.048,-22.909,13.039,178.4661,14.7176,0.0000
C01361=-121.511,-19.067,13.002,177.8637,16.3963,0.0000
C01362=-122.189,-13.416,12.986,178.1457,17.0645,0.0000
C01363=-122.716,-7.050,12.986,178.9750,17.1635,0.0000
C01364=-122.920,0.000,12.986,-179.9999,17.1819,0.0000
C01365=-122.716,7.050,12.986,-178.9751,17.1635,0.0000
C01366=-122.189,13.416,12.986,-178.1458,17.0645,0.0000
C01367=-121.511,19.067,13.002,-177.8637,16.3962,0.0000
C01368=-121.048,22.909,13.039,-178.4661,14.7176,0.0000
C01369=-120.818,25.553,13.086,-179.2525,12.1217,0.0000
C01370=-120.705,27.698,13.130,-179.5784,9.0431,0.0000
C01371=-120.556,29.867,13.161,-179.4158,6.0831,0.0000
C01372=-120.178,32.570,13.176,-179.3657,3.5967,0.0000
C01373=-119.464,35.982,13.183,-179.6066,1.6422,0.0000
C01374=-118.471,39.661,13.189,-179.8748,0.4157,0.0000
C01375=-117.310,43.136,13.196,-179.9743,0.0707,0.0000
C01376=-116.106,46.304,13.199,-179.9968,0.0082,0.0000
C01377=-114.841,49.357,13.199,-179.9965,0.0081,0.0000
C01378=-113.453,52.449,13.196,-179.9682,0.0682,0.0000
C01379=-111.816,55.727,13.189,-179.7945,0.3825,0.0000
C01380=-109.917,59.031,13.183,-179.1168,1.4394,0.0000
C01381=-108.010,61.948,13.176,-177.9029,2.9925,0.0000
C01382=-106.365,64.127,13.161,-176.1015,4.7200,0.0000
C01383=-104.936,65.766,13.130,-173.8735,6.7153,0.0000
C01384=-103.500,67.363,13.086,-171.8818,9.1515,0.0000
C01385=-101.793,69.395,13.039,-170.5301,11.5672,0.0000
C01386=-99.404,72.439,13.002,-169.7025,13.1941,0.0000
C01387=-95.887,76.914,12.986,-169.0120,13.4929,0.0000
C01388=-91.759,81.788,12.986,-168.3741,13.0095,0.0000
C01389=-86.917,86.917,12.986,-167.6668,12.3331,0.0000
C01390=-81.788,91.759,12.986,-166.9906,11.6260,0.0000
C01391=-76.914,95.887,12.986,-166.5072,10.9881,0.0000
C01392=-72.439,99.404,13.002,-166.8059,10.2974,0.0000
C01393=-69.395,101.793,13.039,-168.4328,9.4699,0.0000
C01394=-67.363,103.500,13.086,-170.8485,8.1182,0.0000
C01395=-65.766,104.936,13.130,-173.2847,6.1265,0.0000
C01396=-64.127,106.365,13.161,-175.2800,3.8985,0.0000
C01397=-61.948,108.010,13.176,-177.0075,2.0971,0.0000
C01398=-59.031,109.917,13.183,-178.5606,0.8832,0.0000
C01399=-55.727,111.816,13.189,-179.6175,0.2055,0.0000
C01400=-52.449,113.453,13.196,-179.9318,0.0318,0.0000
C01401=-49.357,114.841,13.199,-179.9919,0.0035,0.0000
C01402=-46.304,116.106,13.199,-179.9918,0.0032,0.0000
C01403=-43.136,117.310,13.196,-179.9293,0.0257,0.0000
C01404=-39.661,118.471,13.189,-179.5843,0.1252,0.0000
C01405=-35.982,119.464,13.183,-178.3578,0.3934,0.0000
C01406=-32.570,120.178,13.176,-176.4033,0.6343,0.0000
C01407=-29.867,120.556,13.161,-173.9169,0.5842,0.0000
C01408=-27.698,120.705,13.130,-170.9569,0.4216,0.0000
C01409=-25.553,120.818,13.086,-167.8783,0.7475,0.0000
C01410=-22.909,121.048,13.039,-165.2824,1.5339,0.0000
C01411=-19.067,121.511,13.002,-163.6038,2.1363,0.0000
C01412=-13.416,122.189,12.986,-162.9355,1.8542,0.0000
C01413=-7.050,122.716,12.986,-162.8365,1.0249,0.0000
C01414=0.000,122.920,12.986,-162.8181,0.0001,0.0000
C01415=0.000,122.228,15.075,-160.5789,0.0001,0.0000
C01416=6.987,122.027,15.074,-160.5994,-1.1667,0.0000
C01417=13.310,121.506,15.075,-160.7077,-2.0797,0.0000
C01418=18.938,120.857,15.098,-161.4419,-2.2356,0.0000
C01419=22.754,120.463,15.154,-163.3609,-1.2202,0.0000
C01420=25.379,120.335,15.225,-166.4251,-0.1124,0.0000
C01421=27.513,120.344,15.292,-170.0054,0.1798,0.0000
C01422=29.672,120.323,15.340,-173.3000,-0.2803,0.0000
C01423=32.360,120.064,15.363,-176.0456,-0.5622,0.0000
C01424=35.784,119.441,15.374,-178.2216,-0.3870,0.0000
C01425=39.505,118.499,15.384,-179.5710,-0.1239,0.0000
C01426=43.038,117.342,15.393,-179.9244,-0.0273,0.0000
C01427=46.271,116.119,15.399,-179.9913,-0.0034,0.0000
C01428=49.390,114.827,15.399,-179.9915,-0.0037,0.0000
C01429=52.541,113.406,15.393,-179.9273,-0.0341,0.0000
C01430=55.857,111.726,15.384,-179.6090,-0.2157,0.0000
C01431=59.154,109.760,15.374,-178.4688,-0.9842,0.0000
C01432=62.016,107.779,15.363,-176.8052,-2.4017,0.0000
C01433=64.100,106.063,15.340,-175.0548,-4.5515,0.0000
C01434=65.641,104.550,15.292,-173.0220,-7.2283,0.0000
C01435=67.144,103.035,15.225,-170.2336,-9.6120,0.0000
C01436=69.091,101.269,15.154,-167.2441,-11.1038,0.0000
C01437=72.068,98.850,15.098,-165.1580,-11.8482,0.0000
C01438=76.506,95.329,15.075,-164.7199,-12.5080,0.0000
C01439=81.346,91.227,15.074,-165.2423,-13.2039,0.0000
C01440=86.429,86.429,15.075,-166.0013,-13.9988,0.0000
C01441=91.227,81.346,15.074,-166.7961,-14.7576,0.0000
C01442=95.329,76.506,15.075,-167.4919,-15.2800,0.0000
C01443=98.850,72.068,15.098,-168.1519,-14.8421,0.0000
C01444=101.269,69.091,15.154,-168.8962,-12.7559,0.0000
C01445=103.035,67.144,15.225,-170.3880,-9.7664,0.0000
C01446=104.550,65.641,15.292,-172.7717,-6.9780,0.0000
C01447=106.063,64.100,15.340,-175.4485,-4.9452,0.0000
C01448=107.779,62.016,15.363,-177.5983,-3.1948,0.0000
C01449=109.760,59.154,15.374,-179.0158,-1.5312,0.0000
C01450=111.726,55.857,15.384,-179.7843,-0.3910,0.0000
C01451=113.406,52.541,15.393,-179.9659,-0.0727,0.0000
C01452=114.827,49.390,15.399,-179.9963,-0.0085,0.0000
C01453=116.119,46.271,15.399,-179.9966,-0.0087,0.0000
C01454=117.342,43.038,15.393,-179.9727,-0.0756,0.0000
C01455=118.499,39.505,15.384,-179.8761,-0.4290,0.0000
C01456=119.441,35.784,15.374,-179.6130,-1.7784,0.0000
C01457=120.064,32.360,15.363,-179.4378,-3.9544,0.0000
C01458=120.323,29.672,15.340,-179.7197,-6.7000,0.0000
C01459=120.344,27.513,15.292,179.8202,-9.9946,0.0000
C01460=120.335,25.379,15.225,-179.8876,-13.5749,0.0000
C01461=120.463,22.754,15.154,-178.7798,-16.6391,0.0000
C01462=120.857,18.938,15.098,-177.7644,-18.5581,0.0000
C01463=121.506,13.310,15.075,-177.9203,-19.2923,0.0000
C01464=122.027,6.987,15.074,-178.8333,-19.4006,0.0000
C01465=122.228,0.000,15.075,179.9999,-19.4211,0.0000
C01466=122.027,-6.987,15.074,178.8334,-19.4006,0.0000
C01467=121.506,-13.310,15.075,177.9205,-19.2923,0.0000
C01468=120.857,-18.938,15.098,177.7643,-18.5581,0.0000
C01469=120.463,-22.754,15.154,178.7798,-16.6391,0.0000
C01470=120.335,-25.379,15.225,179.8876,-13.5749,0.0000
C01471=120.344,-27.513,15.292,-179.8202,-9.9946,0.0000
C01472=120.323,-29.672,15.340,179.7197,-6.7000,0.0000
C01473=120.064,-32.360,15.363,179.4378,-3.9544,0.0000
C01474=119.441,-35.784,15.374,179.6130,-1.7784,0.0000
C01475=118.499,-39.505,15.384,179.8761,-0.4290,0.0000
C01476=117.342,-43.038,15.393,179.9727,-0.0756,0.0000
C01477=116.119,-46.271,15.399,179.9966,-0.0087,0.0000
C01478=114.827,-49.390,15.399,179.9963,-0.0085,0.0000
C01479=113.406,-52.541,15.393,179.9659,-0.0727,0.0000
C01480=111.726,-55.857,15.384,179.7843,-0.3910,0.0000
C01481=109.760,-59.154,15.374,179.0158,-1.5312,0.0000
C01482=107.779,-62.016,15.363,177.5983,-3.1948,0.0000
C01483=106.063,-64.100,15.340,175.4485,-4.9452,0.0000
C01484=104.550,-65.641,15.292,172.7717,-6.9780,0.0000
C01485=103.035,-67.144,15.225,170.3880,-9.7664,0.0000
C01486=101.269,-69.091,15.154,168.8962,-12.7559,0.0000
C01487=98.850,-72.068,15.098,168.1518,-14.8420,0.0000
C01488=95.329,-76.506,15.075,167.4920,-15.2801,0.0000
C01489=91.227,-81.346,15.074,166.7961,-14.7577,0.0000
C01490=86.429,-86.429,15.075,166.0012,-13.9987,0.0000
C01491=81.346,-91.227,15.074,165.2424,-13.2039,0.0000
C01492=76.506,-95.329,15.075,164.7200,-12.5081,0.0000
C01493=72.068,-98.850,15.098,165.1579,-11.8481,0.0000
C01494=69.091,-101.269,15.154,167.2441,-11.1038,0.0000
C01495=67.144,-103.035,15.225,170.2336,-9.6120,0.0000
C01496=65.641,-104.550,15.292,173.0220,-7.2283,0.0000
C01497=64.100,-106.063,15.340,175.0548,-4.5515,0.0000
C01498=62.016,-107.779,15.363,176.8052,-2.4017,0.0000
C01499=59.154,-109.760,15.374,178.4688,-0.9842,0.0000
C01500=55.857,-111.726,15.384,179.6090,-0.2157,0.0000
C01501=52.541,-113.406,15.393,179.9273,-0.0341,0.0000
C01502=49.390,-114.827,15.399,179.9915,-0.0037,0.0000
C01503=46.271,-116.119,15.399,179.9913,-0.0034,0.0000
C01504=43.038,-117.342,15.393,179.9244,-0.0273,0.0000
C01505=39.505,-118.499,15.384,179.5710,-0.1239,0.0000
C01506=35.784,-119.441,15.374,178.2216,-0.3870,0.0000
C01507=32.360,-120.064,15.363,176.0456,-0.5622,0.0000
C01508=29.672,-120.323,15.340,173.3000,-0.2803,0.0000
C01509=27.513,-120.344,15.292,170.0054,0.1798,0.0000
C01510=25.379,-120.335,15.225,166.4251,-0.1124,0.0000
C01511=22.754,-120.463,15.154,163.3609,-1.2202,0.0000
C01512=18.938,-120.857,15.098,161.4419,-2.2356,0.0000
C01513=13.310,-121.506,15.075,160.7077,-2.0797,0.0000
C01514=6.987,-122.027,15.074,160.5994,-1.1667,0.0000
C01515=0.000,-122.228,15.075,160.5789,0.0001,0.0000
C01516=0.000,-122.228,15.075,160.5789,0.0001,0.0000
C01517=-6.987,-122.027,15.074,160.5994,1.1666,0.0000
C01518=-13.310,-121.506,15.075,160.7077,2.0795,0.0000
C01519=-18.938,-120.857,15.098,161.4419,2.2357,0.0000
C01520=-22.754,-120.463,15.154,163.3609,1.2202,0.0000
C01521=-25.379,-120.335,15.225,166.4251,0.1124,0.0000
C01522=-27.513,-120.344,15.292,170.0054,-0.1798,0.0000
C01523=-29.672,-120.323,15.340,173.3000,0.2803,0.0000
C01524=-32.360,-120.064,15.363,176.0456,0.5622,0.0000
C01525=-35.784,-119.441,15.374,178.2216,0.3870,0.0000
C01526=-39.505,-118.499,15.384,179.5710,0.1239,0.0000
C01527=-43.038,-117.342,15.393,179.9244,0.0273,0.0000
C01528=-46.271,-116.119,15.399,179.9913,0.0034,0.0000
C01529=-49.390,-114.827,15.399,179.9915,0.0037,0.0000
C01530=-52.541,-113.406,15.393,179.9273,0.0341,0.0000
C01531=-55.857,-111.726,15.384,179.6090,0.2157,0.0000
C01532=-59.154,-109.760,15.374,178.4688,0.9842,0.0000
C01533=-62.016,-107.779,15.363,176.8052,2.4017,0.0000
C01534=-64.100,-106.063,15.340,175.0548,4.5515,0.0000
C01535=-65.641,-104.550,15.292,173.0220,7.2283,0.0000
C01536=-67.144,-103.035,15.225,170.2336,9.6120,0.0000
C01537=-69.091,-101.269,15.154,167.2441,11.1038,0.0000
C01538=-72.068,-98.850,15.098,165.1580,11.8482,0.0000
C01539=-76.506,-95.329,15.075,164.7199,12.5080,0.0000
C01540=-81.346,-91.227,15.074,165.2423,13.2039,0.0000
C01541=-86.429,-86.429,15.075,166.0013,13.9988,0.0000
C01542=-91.227,-81.346,15.074,166.7961,14.7576,0.0000
C01543=-95.329,-76.506,15.075,167.4919,15.2800,0.0000
C01544=-98.850,-72.068,15.098,168.1519,14.8421,0.0000
C01545=-101.269,-69.091,15.154,168.8962,12.7559,0.0000
C01546=-103.035,-67.144,15.225,170.3880,9.7664,0.0000
C01547=-104.550,-65.641,15.292,172.7717,6.9780,0.0000
C01548=-106.063,-64.100,15.340,175.4485,4.9452,0.0000
C01549=-107.779,-62.016,15.363,177.5983,3.1948,0.0000
C01550=-109.760,-59.154,15.374,179.0158,1.5312,0.0000
C01551=-111.726,-55.857,15.384,179.7843,0.3910,0.0000
C01552=-113.406,-52.541,15.393,179.9659,0.0727,0.0000
C01553=-114.827,-49.390,15.399,179.9963,0.0085,0.0000
C01554=-116.119,-46.271,15.399,179.9966,0.0087,0.0000
C01555=-117.342,-43.038,15.393,179.9727,0.0756,0.0000
C01556=-118.499,-39.505,15.384,179.8761,0.4290,0.0000
C01557=-119.441,-35.784,15.374,179.6130,1.7784,0.0000
C01558=-120.064,-32.360,15.363,179.4378,3.9544,0.0000
C01559=-120.323,-29.672,15.340,179.7197,6.7000,0.0000
C01560=-120.344,-27.513,15.292,-179.8202,9.9946,0.0000
C01561=-120.335,-25.379,15.225,179.8876,13.5749,0.0000
C01562=-120.463,-22.754,15.154,178.7798,16.6391,0.0000
C01563=-120.857,-18.938,15.098,177.7644,18.5581,0.0000
C01564=-121.506,-13.310,15.075,177.9203,19.2923,0.0000
C01565=-122.027,-6.987,15.074,178.8333,19.4006,0.0000
C01566=-122.228,0.000,15.075,-179.9999,19.4211,0.0000
C01567=-122.027,6.987,15.074,-178.8334,19.4006,0.0000
C01568=-121.506,13.310,15.075,-177.9205,19.2923,0.0000
C01569=-120.857,18.938,15.098,-177.7643,18.5581,0.0000
C01570=-120.463,22.754,15.154,-178.7798,16.6391,0.0000
C01571=-120.335,25.379,15.225,-179.8876,13.5749,0.0000
C01572=-120.344,27.513,15.292,179.8202,9.9946,0.0000
C01573=-120.323,29.672,15.340,-179.7197,6.7000,0.0000
C01574=-120.064,32.360,15.363,-179.4378,3.9544,0.0000
C01575=-119.441,35.784,15.374,-179.6130,1.7784,0.0000
C01576=-118.499,39.505,15.384,-179.8761,0.4290,0.0000
C01577=-117.342,43.038,15.393,-179.9727,0.0756,0.0000
C01578=-116.119,46.271,15.399,-179.9966,0.0087,0.0000
C01579=-114.827,49.390,15.399,-179.9963,0.0085,0.0000
C01580=-113.406,52.541,15.393,-179.9659,0.0727,0.0000
C01581=-111.726,55.857,15.384,-179.7843,0.3910,0.0000
C01582=-109.760,59.154,15.374,-179.0158,1.5312,0.0000
C01583=-107.779,62.016,15.363,-177.5983,3.1948,0.0000
C01584=-106.063,64.100,15.340,-175.4485,4.9452,0.0000
C01585=-104.550,65.641,15.292,-172.7717,6.9780,0.0000
C01586=-103.035,67.144,15.225,-170.3880,9.7664,0.0000
C01587=-101.269,69.091,15.154,-168.8962,12.7559,0.0000
C01588=-98.850,72.068,15.098,-168.1518,14.8420,0.0000
C01589=-95.329,76.506,15.075,-167.4920,15.2801,0.0000
C01590=-91.227,81.346,15.074,-166.7961,14.7577,0.0000
C01591=-86.429,86.429,15.075,-166.0012,13.9987,0.0000
C01592=-81.346,91.227,15.074,-165.2424,13.2039,0.0000
C01593=-76.506,95.329,15.075,-164.7200,12.5081,0.0000
C01594=-72.068,98.850,15.098,-165.1579,11.8481,0.0000
C01595=-69.091,101.269,15.154,-167.2441,11.1038,0.0000
C01596=-67.144,103.035,15.225,-170.2336,9.6120,0.0000
C01597=-65.641,104.550,15.292,-173.0220,7.2283,0.0000
C01598=-64.100,106.063,15.340,-175.0548,4.5515,0.0000
C01599=-62.016,107.779,15.363,-176.8052,2.4017,0.0000
C01600=-59.154,109.760,15.374,-178.4688,0.9842,0.0000
C01601=-55.857,111.726,15.384,-179.6090,0.2157,0.0000
C01602=-52.541,113.406,15.393,-179.9273,0.0341,0.0000
C01603=-49.390,114.827,15.399,-179.9915,0.0037,0.0000
C01604=-46.271,116.119,15.399,-179.9913,0.0034,0.0000
C01605=-43.038,117.342,15.393,-179.9244,0.0273,0.0000
C01606=-39.505,118.499,15.384,-179.5710,0.1239,0.0000
C01607=-35.784,119.441,15.374,-178.2216,0.3870,0.0000
C01608=-32.360,120.064,15.363,-176.0456,0.5622,0.0000
C01609=-29.672,120.323,15.340,-173.3000,0.2803,0.0000
C01610=-27.513,120.344,15.292,-170.0054,-0.1798,0.0000
C01611=-25.379,120.335,15.225,-166.4251,0.1124,0.0000
C01612=-22.754,120.463,15.154,-163.3609,1.2202,0.0000
C01613=-18.938,120.857,15.098,-161.4419,2.2357,0.0000
C01614=-13.310,121.506,15.075,-160.7077,2.0795,0.0000
C01615=-6.987,122.027,15.074,-160.5994,1.1666,0.0000
C01616=0.000,122.228,15.075,-160.5789,0.0001,0.0000
C01617=0.000,121.459,17.136,-158.5165,0.0001,0.0000
C01618=6.917,121.260,17.135,-158.5388,-1.3000,0.0000
C01619=13.191,120.746,17.136,-158.6546,-2.2779,0.0000
C01620=18.794,120.128,17.169,-159.4470,-2.2431,0.0000
C01621=22.580,119.809,17.247,-161.6340,-0.6924,0.0000
C01622=25.184,119.793,17.348,-165.2455,0.7774,0.0000
C01623=27.305,119.938,17.444,-169.3441,0.9740,0.0000
C01624=29.452,120.062,17.513,-172.8760,0.1423,0.0000
C01625=32.122,119.934,17.546,-175.7883,-0.4355,0.0000
C01626=35.561,119.414,17.563,-178.1363,-0.3602,0.0000
C01627=39.328,118.531,17.576,-179.5773,-0.1164,0.0000
C01628=42.927,117.379,17.590,-179.9218,-0.0280,0.0000
C01629=46.233,116.133,17.599,-179.9911,-0.0035,0.0000
C01630=49.427,114.811,17.599,-179.9912,-0.0038,0.0000
C01631=52.646,113.353,17.590,-179.9249,-0.0354,0.0000
C01632=56.005,111.623,17.576,-179.6188,-0.2166,0.0000
C01633=59.293,109.584,17.563,-178.4274,-1.0635,0.0000
C01634=62.093,107.520,17.546,-176.7121,-2.6736,0.0000
C01635=64.071,105.722,17.513,-175.0494,-5.1502,0.0000
C01636=65.501,104.117,17.444,-173.0994,-8.2542,0.0000
C01637=66.899,102.515,17.348,-169.9831,-11.0794,0.0000
C01638=68.751,100.685,17.247,-166.3254,-12.7464,0.0000
C01639=71.654,98.232,17.169,-163.6790,-13.3562,0.0000
C01640=76.053,94.708,17.136,-163.0665,-13.9395,0.0000
C01641=80.853,90.635,17.135,-163.6151,-14.6781,0.0000
C01642=85.885,85.885,17.136,-164.4481,-15.5520,0.0000
C01643=90.635,80.853,17.135,-165.3218,-16.3848,0.0000
C01644=94.708,76.053,17.136,-166.0603,-16.9334,0.0000
C01645=98.232,71.654,17.169,-166.6439,-16.3210,0.0000
C01646=100.685,68.751,17.247,-167.2536,-13.6746,0.0000
C01647=102.515,66.899,17.348,-168.9206,-10.0169,0.0000
C01648=104.117,65.501,17.444,-171.7458,-6.9006,0.0000
C01649=105.722,64.071,17.513,-174.8498,-4.9506,0.0000
C01650=107.520,62.093,17.546,-177.3264,-3.2879,0.0000
C01651=109.584,59.293,17.563,-178.9365,-1.5726,0.0000
C01652=111.623,56.005,17.576,-179.7834,-0.3812,0.0000
C01653=113.353,52.646,17.590,-179.9646,-0.0751,0.0000
C01654=114.811,49.427,17.599,-179.9962,-0.0088,0.0000
C01655=116.133,46.233,17.599,-179.9965,-0.0089,0.0000
C01656=117.379,42.927,17.590,-179.9720,-0.0782,0.0000
C01657=118.531,39.328,17.576,-179.8836,-0.4227,0.0000
C01658=119.414,35.561,17.563,-179.6398,-1.8637,0.0000
C01659=119.934,32.122,17.546,-179.5645,-4.2117,0.0000
C01660=120.062,29.452,17.513,179.8577,-7.1240,0.0000
C01661=119.938,27.305,17.444,179.0260,-10.6559,0.0000
C01662=119.793,25.184,17.348,179.2226,-14.7545,0.0000
C01663=119.809,22.580,17.247,-179.3076,-18.3660,0.0000
C01664=120.128,18.794,17.169,-177.7569,-20.5530,0.0000
C01665=120.746,13.191,17.136,-177.7221,-21.3454,0.0000
C01666=121.260,6.917,17.135,-178.7000,-21.4612,0.0000
C01667=121.459,0.000,17.136,179.9999,-21.4835,0.0000
C01668=121.260,-6.916,17.135,178.7002,-21.4611,0.0000
C01669=120.746,-13.191,17.136,177.7223,-21.3454,0.0000
C01670=120.128,-18.794,17.169,177.7568,-20.5529,0.0000
C01671=119.809,-22.580,17.247,179.3076,-18.3660,0.0000
C01672=119.793,-25.184,17.348,-179.2226,-14.7545,0.0000
C01673=119.938,-27.305,17.444,-179.0260,-10.6559,0.0000
C01674=120.062,-29.452,17.513,-179.8577,-7.1240,0.0000
C01675=119.934,-32.122,17.546,179.5645,-4.2117,0.0000
C01676=119.414,-35.561,17.563,179.6398,-1.8637,0.0000
C01677=118.531,-39.328,17.576,179.8836,-0.4227,0.0000
C01678=117.379,-42.927,17.590,179.9720,-0.0782,0.0000
C01679=116.133,-46.233,17.599,179.9965,-0.0089,0.0000
C01680=114.811,-49.427,17.599,179.9962,-0.0088,0.0000
C01681=113.353,-52.646,17.590,179.9646,-0.0751,0.0000
C01682=111.623,-56.005,17.576,179.7834,-0.3812,0.0000
C01683=109.584,-59.293,17.563,178.9365,-1.5726,0.0000
C01684=107.520,-62.093,17.546,177.3264,-3.2879,0.0000
C01685=105.722,-64.071,17.513,174.8498,-4.9506,0.0000
C01686=104.117,-65.501,17.444,171.7458,-6.9006,0.0000
C01687=102.515,-66.899,17.348,168.9206,-10.0169,0.0000
C01688=100.685,-68.751,17.247,167.2536,-13.6746,0.0000
C01689=98.232,-71.654,17.169,166.6438,-16.3210,0.0000
C01690=94.708,-76.053,17.136,166.0605,-16.9335,0.0000
C01691=90.635,-80.853,17.135,165.3219,-16.3849,0.0000
C01692=85.885,-85.885,17.136,164.4480,-15.5519,0.0000
C01693=80.853,-90.635,17.135,163.6152,-14.6782,0.0000
C01694=76.053,-94.708,17.136,163.0666,-13.9397,0.0000
C01695=71.654,-98.232,17.169,163.6790,-13.3561,0.0000
C01696=68.751,-100.685,17.247,166.3254,-12.7464,0.0000
C01697=66.899,-102.515,17.348,169.9831,-11.0794,0.0000
C01698=65.501,-104.117,17.444,173.0994,-8.2542,0.0000
C01699=64.071,-105.722,17.513,175.0494,-5.1502,0.0000
C01700=62.093,-107.520,17.546,176.7121,-2.6736,0.0000
C01701=59.293,-109.584,17.563,178.4274,-1.0635,0.0000
C01702=56.005,-111.623,17.576,179.6188,-0.2166,0.0000
C01703=52.646,-113.353,17.590,179.9249,-0.0354,0.0000
C01704=49.427,-114.811,17.599,179.9912,-0.0038,0.0000
C01705=46.233,-116.133,17.599,179.9911,-0.0035,0.0000
C01706=42.927,-117.379,17.590,179.9218,-0.0280,0.0000
C01707=39.328,-118.531,17.576,179.5773,-0.1164,0.0000
C01708=35.561,-119.414,17.563,178.1363,-0.3602,0.0000
C01709=32.122,-119.934,17.546,175.7883,-0.4355,0.0000
C01710=29.452,-120.062,17.513,172.8760,0.1423,0.0000
C01711=27.305,-119.938,17.444,169.3441,0.9740,0.0000
C01712=25.184,-119.793,17.348,165.2455,0.7774,0.0000
C01713=22.580,-119.809,17.247,161.6340,-0.6924,0.0000
C01714=18.794,-120.128,17.169,159.4470,-2.2431,0.0000
C01715=13.191,-120.746,17.136,158.6546,-2.2779,0.0000
C01716=6.917,-121.260,17.135,158.5388,-1.3000,0.0000
C01717=0.000,-121.459,17.136,158.5165,0.0001,0.0000
C01718=0.000,-121.459,17.136,158.5165,0.0001,0.0000
C01719=-6.916,-121.260,17.135,158.5389,1.2998,0.0000
C01720=-13.191,-120.746,17.136,158.6546,2.2777,0.0000
C01721=-18.794,-120.128,17.169,159.4471,2.2432,0.0000
C01722=-22.580,-119.809,17.247,161.6340,0.6924,0.0000
C01723=-25.184,-119.793,17.348,165.2455,-0.7774,0.0000
C01724=-27.305,-119.938,17.444,169.3441,-0.9740,0.0000
C01725=-29.452,-120.062,17.513,172.8760,-0.1423,0.0000
C01726=-32.122,-119.934,17.546,175.7883,0.4355,0.0000
C01727=-35.561,-119.414,17.563,178.1363,0.3602,0.0000
C01728=-39.328,-118.531,17.576,179.5773,0.1164,0.0000
C01729=-42.927,-117.379,17.590,179.9218,0.0280,0.0000
C01730=-46.233,-116.133,17.599,179.9911,0.0035,0.0000
C01731=-49.427,-114.811,17.599,179.9912,0.0038,0.0000
C01732=-52.646,-113.353,17.590,179.9249,0.0354,0.0000
C01733=-56.005,-111.623,17.576,179.6188,0.2166,0.0000
C01734=-59.293,-109.584,17.563,178.4274,1.0635,0.0000
C01735=-62.093,-107.520,17.546,176.7121,2.6736,0.0000
C01736=-64.071,-105.722,17.513,175.0494,5.1502,0.0000
C01737=-65.501,-104.117,17.444,173.0994,8.2542,0.0000
C01738=-66.899,-102.515,17.348,169.9831,11.0794,0.0000
C01739=-68.751,-100.685,17.247,166.3254,12.7464,0.0000
C01740=-71.654,-98.232,17.169,163.6790,13.3562,0.0000
C01741=-76.053,-94.708,17.136,163.0665,13.9395,0.0000
C01742=-80.853,-90.635,17.135,163.6151,14.6781,0.0000
C01743=-85.885,-85.885,17.136,164.4481,15.5520,0.0000
C01744=-90.635,-80.853,17.135,165.3218,16.3848,0.0000
C01745=-94.708,-76.053,17.136,166.0603,16.9334,0.0000
C01746=-98.232,-71.654,17.169,166.6439,16.3210,0.0000
C01747=-100.685,-68.751,17.247,167.2536,13.6746,0.0000
C01748=-102.515,-66.899,17.348,168.9206,10.0169,0.0000
C01749=-104.117,-65.501,17.444,171.7458,6.9006,0.0000
C01750=-105.722,-64.071,17.513,174.8498,4.9506,0.0000
C01751=-107.520,-62.093,17.546,177.3264,3.2879,0.0000
C01752=-109.584,-59.293,17.563,178.9365,1.5726,0.0000
C01753=-111.623,-56.005,17.576,179.7834,0.3812,0.0000
C01754=-113.353,-52.646,17.590,179.9646,0.0751,0.0000
C01755=-114.811,-49.427,17.599,179.9962,0.0088,0.0000
C01756=-116.133,-46.233,17.599,179.9965,0.0089,0.0000
C01757=-117.379,-42.927,17.590,179.9720,0.0782,0.0000
C01758=-118.531,-39.328,17.576,179.8836,0.4227,0.0000
C01759=-119.414,-35.561,17.563,179.6398,1.8637,0.0000
C01760=-119.934,-32.122,17.546,179.5645,4.2117,0.0000
C01761=-120.062,-29.452,17.513,-179.8577,7.1240,0.0000
C01762=-119.938,-27.305,17.444,-179.0260,10.6559,0.0000
C01763=-119.793,-25.184,17.348,-179.2226,14.7545,0.0000
C01764=-119.809,-22.580,17.247,179.3076,18.3660,0.0000
C01765=-120.128,-18.794,17.169,177.7569,20.5530,0.0000
C01766=-120.746,-13.191,17.136,177.7221,21.3454,0.0000
C01767=-121.260,-6.917,17.135,178.7000,21.4612,0.0000
C01768=-121.459,0.000,17.136,-179.9999,21.4835,0.0000
C01769=-121.260,6.916,17.135,-178.7002,21.4611,0.0000
C01770=-120.746,13.191,17.136,-177.7223,21.3454,0.0000
C01771=-120.128,18.794,17.169,-177.7568,20.5529,0.0000
C01772=-119.809,22.580,17.247,-179.3076,18.3660,0.0000
C01773=-119.793,25.184,17.348,179.2226,14.7545,0.0000
C01774=-119.938,27.305,17.444,179.0260,10.6559,0.0000
C01775=-120.062,29.452,17.513,179.8577,7.1240,0.0000
C01776=-119.934,32.122,17.546,-179.5645,4.2117,0.0000
C01777=-119.414,35.561,17.563,-179.6398,1.8637,0.0000
C01778=-118.531,39.328,17.576,-179.8836,0.4227,0.0000
C01779=-117.379,42.927,17.590,-179.9720,0.0782,0.0000
C01780=-116.133,46.233,17.599,-179.9965,0.0089,0.0000
C01781=-114.811,49.427,17.599,-179.9962,0.0088,0.0000
C01782=-113.353,52.646,17.590,-179.9646,0.0751,0.0000
C01783=-111.623,56.005,17.576,-179.7834,0.3812,0.0000
C01784=-109.584,59.293,17.563,-178.9365,1.5726,0.0000
C01785=-107.520,62.093,17.546,-177.3264,3.2879,0.0000
C01786=-105.722,64.071,17.513,-174.8498,4.9506,0.0000
C01787=-104.117,65.501,17.444,-171.7458,6.9006,0.0000
C01788=-102.515,66.899,17.348,-168.9206,10.0169,0.0000
C01789=-100.685,68.751,17.247,-167.2536,13.6746,0.0000
C01790=-98.232,71.654,17.169,-166.6438,16.3210,0.0000
C01791=-94.708,76.053,17.136,-166.0605,16.9335,0.0000
C01792=-90.635,80.853,17.135,-165.3219,16.3849,0.0000
C01793=-85.885,85.885,17.136,-164.4480,15.5519,0.0000
C01794=-80.853,90.635,17.135,-163.6152,14.6782,0.0000
C01795=-76.053,94.708,17.136,-163.0666,13.9397,0.0000
C01796=-71.654,98.232,17.169,-163.6790,13.3561,0.0000
C01797=-68.751,100.685,17.247,-166.3254,12.7464,0.0000
C01798=-66.899,102.515,17.348,-169.9831,11.0794,0.0000
C01799=-65.501,104.117,17.444,-173.0994,8.2542,0.0000
C01800=-64.071,105.722,17.513,-175.0494,5.1502,0.0000
C01801=-62.093,107.520,17.546,-176.7121,2.6736,0.0000
C01802=-59.293,109.584,17.563,-178.4274,1.0635,0.0000
C01803=-56.005,111.623,17.576,-179.6188,0.2166,0.0000
C01804=-52.646,113.353,17.590,-179.9249,0.0354,0.0000
C01805=-49.427,114.811,17.599,-179.9912,0.0038,0.0000
C01806=-46.233,116.133,17.599,-179.9911,0.0035,0.0000
C01807=-42.927,117.379,17.590,-179.9218,0.0280,0.0000
C01808=-39.328,118.531,17.576,-179.5773,0.1164,0.0000
C01809=-35.561,119.414,17.563,-178.1363,0.3602,0.0000
C01810=-32.122,119.934,17.546,-175.7883,0.4355,0.0000
C01811=-29.452,120.062,17.513,-172.8760,-0.1423,0.0000
C01812=-27.305,119.938,17.444,-169.3441,-0.9740,0.0000
C01813=-25.184,119.793,17.348,-165.2455,-0.7774,0.0000
C01814=-22.580,119.809,17.247,-161.6340,0.6924,0.0000
C01815=-18.794,120.128,17.169,-159.4471,2.2432,0.0000
C01816=-13.191,120.746,17.136,-158.6546,2.2777,0.0000
C01817=-6.916,121.260,17.135,-158.5389,1.2998,0.0000
C01818=0.000,121.459,17.136,-158.5165,0.0001,0.0000
C01819=0.000,120.619,19.169,-156.6224,0.0002,0.0000
C01820=6.840,120.423,19.168,-156.6463,-1.4248,0.0000
C01821=13.062,119.916,19.170,-156.7679,-2.4488,0.0000
C01822=18.637,119.331,19.213,-157.6149,-2.1561,0.0000
C01823=22.390,119.093,19.319,-160.1217,0.0530,0.0000
C01824=24.970,119.198,19.455,-164.3916,1.8868,0.0000
C01825=27.076,119.491,19.586,-169.0248,1.9005,0.0000
C01826=29.209,119.772,19.680,-172.6791,0.6529,0.0000
C01827=31.859,119.791,19.725,-175.6434,-0.2625,0.0000
C01828=35.314,119.384,19.749,-178.1045,-0.3162,0.0000
C01829=39.133,118.567,19.767,-179.6035,-0.1035,0.0000
C01830=42.803,117.420,19.786,-179.9215,-0.0280,0.0000
C01831=46.191,116.149,19.798,-179.9912,-0.0035,0.0000
C01832=49.468,114.792,19.798,-179.9913,-0.0038,0.0000
C01833=52.762,113.295,19.786,-179.9247,-0.0358,0.0000
C01834=56.168,111.510,19.767,-179.6465,-0.2072,0.0000
C01835=59.447,109.388,19.749,-178.4360,-1.1171,0.0000
C01836=62.177,107.232,19.725,-176.7314,-2.8984,0.0000
C01837=64.038,105.345,19.680,-175.2675,-5.6483,0.0000
C01838=65.347,103.638,19.586,-173.5152,-9.1234,0.0000
C01839=66.629,101.942,19.455,-170.1157,-12.4530,0.0000
C01840=68.379,100.044,19.319,-165.6938,-14.3765,0.0000
C01841=71.201,97.558,19.213,-162.3669,-14.8215,0.0000
C01842=75.557,94.030,19.170,-161.5422,-15.2854,0.0000
C01843=80.315,89.988,19.168,-162.1046,-16.0519,0.0000
C01844=85.291,85.291,19.169,-163.0036,-16.9966,0.0000
C01845=89.988,80.316,19.168,-163.9480,-17.8952,0.0000
C01846=94.030,75.557,19.170,-164.7144,-18.4576,0.0000
C01847=97.558,71.201,19.213,-165.1787,-17.6332,0.0000
C01848=100.044,68.379,19.319,-165.6235,-14.3062,0.0000
C01849=101.942,66.629,19.455,-167.5470,-9.8843,0.0000
C01850=103.638,65.347,19.586,-170.8766,-6.4848,0.0000
C01851=105.345,64.038,19.680,-174.3517,-4.7325,0.0000
C01852=107.232,62.177,19.725,-177.1016,-3.2686,0.0000
C01853=109.388,59.447,19.749,-178.8829,-1.5640,0.0000
C01854=111.510,56.168,19.767,-179.7928,-0.3535,0.0000
C01855=113.295,52.762,19.786,-179.9642,-0.0753,0.0000
C01856=114.792,49.468,19.798,-179.9962,-0.0087,0.0000
C01857=116.149,46.191,19.798,-179.9965,-0.0088,0.0000
C01858=117.420,42.803,19.786,-179.9720,-0.0785,0.0000
C01859=118.567,39.133,19.767,-179.8965,-0.3965,0.0000
C01860=119.384,35.314,19.749,-179.6838,-1.8955,0.0000
C01861=119.791,31.859,19.725,-179.7375,-4.3566,0.0000
C01862=119.772,29.209,19.680,179.3471,-7.3209,0.0000
C01863=119.491,27.076,19.586,178.0995,-10.9752,0.0000
